LIN {X 0,Y 518.163,Z 728.095,A -85,B 0,C 180,E1 -4999.763,E2 -4999.763} C_VEL
LIN {X 0,Y 517.896,Z 738.556,A -85,B 0,C 180,E1 -5000.474,E2 -5000.474} C_VEL
LIN {X 0,Y 517.639,Z 748.894,A -85,B 0,C 180,E1 -5001.351,E2 -5001.351} C_VEL
LIN {X 0,Y 517.372,Z 758.155,A -85,B 0,C 180,E1 -5002.317,E2 -5002.317} C_VEL
LIN {X 0,Y 517.046,Z 767.447,A -85,B 0,C 180,E1 -5003.531,E2 -5003.531} C_VEL
LIN {X 0,Y 516.894,Z 774.412,A -85,B 0,C 180,E1 -5004.667,E2 -5004.667} C_VEL
LIN {X 0,Y 516.72,Z 779.315,A -85,B 0,C 180,E1 -5005.636,E2 -5005.636} C_VEL
LIN {X 0,Y 516.615,Z 783.22,A -85,B 0,C 180,E1 -5006.567,E2 -5006.567} C_VEL
LIN {X 0,Y 516.59,Z 786.474,A -85,B 0,C 180,E1 -5007.511,E2 -5007.511} C_VEL
LIN {X 0,Y 516.499,Z 789.918,A -85,B 0,C 180,E1 -5008.864,E2 -5008.864} C_VEL
LIN {X 0,Y 516.448,Z 791.553,A -85,B 0,C 180,E1 -5009.767,E2 -5009.767} C_VEL
LIN {X 0,Y 516.407,Z 792.613,A -85,B 0,C 180,E1 -5010.663,E2 -5010.663} C_VEL
LIN {X 0,Y 516.396,Z 793.257,A -85,B 0,C 180,E1 -5012.207,E2 -5012.207} C_VEL
LIN {X 0,Y 516.435,Z 792.788,A -85,B 0,C 180,E1 -5013.315,E2 -5013.315} C_VEL
LIN {X 0,Y 516.442,Z 791.847,A -85,B 0,C 180,E1 -5014.184,E2 -5014.184} C_VEL
LIN {X 0,Y 516.562,Z 789.005,A -85,B 0,C 180,E1 -5015.722,E2 -5015.722} C_VEL
LIN {X 0,Y 516.653,Z 784.693,A -85,B 0,C 180,E1 -5017.189,E2 -5017.189} C_VEL
LIN {X 0,Y 516.772,Z 779.621,A -85,B 0,C 180,E1 -5018.457,E2 -5018.457} C_VEL
LIN {X 0,Y 516.959,Z 774.001,A -85,B 0,C 180,E1 -5019.569,E2 -5019.569} C_VEL
LIN {X 0,Y 517.22,Z 766.534,A -85,B 0,C 180,E1 -5020.761,E2 -5020.761} C_VEL
LIN {X 0,Y 517.462,Z 757.238,A -85,B 0,C 180,E1 -5021.938,E2 -5021.938} C_VEL
LIN {X 0,Y 517.742,Z 747.459,A -85,B 0,C 180,E1 -5022.93,E2 -5022.93} C_VEL
LIN {X 0,Y 518.011,Z 737.439,A -85,B 0,C 180,E1 -5023.75,E2 -5023.75} C_VEL
LIN {X 0,Y 518.228,Z 727.164,A -85,B 0,C 180,E1 -5024.43,E2 -5024.43} C_VEL
LIN {X 0,Y 518.371,Z 718.099,A -85,B 0,C 180,E1 -5024.913,E2 -5024.913} C_VEL
LIN {X 0,Y 516.951,Z 712.094,A -85,B 0,C 180,E1 -5025.232,E2 -5025.232} C_VEL
LIN {X 0,Y 516.971,Z 712.089,A -85,B 0,C 180,E1 -5028.234,E2 -5028.234} C_VEL
LIN {X 0,Y 516.968,Z 712.091,A -85,B 0,C 180,E1 -5031.4,E2 -5031.4} C_VEL
LIN {X 0,Y 517.017,Z 712.078,A -85,B 0,C 180,E1 -5034.54,E2 -5034.54} C_VEL
LIN {X 0,Y 517.085,Z 712.078,A -85,B 0,C 180,E1 -5037.663,E2 -5037.663} C_VEL
LIN {X 0,Y 517.095,Z 712.068,A -85,B 0,C 180,E1 -5040.779,E2 -5040.779} C_VEL
LIN {X 0,Y 516.988,Z 712.08,A -85,B 0,C 180,E1 -5043.117,E2 -5043.117} C_VEL
LIN {X 0,Y 517.013,Z 712.083,A -85,B 0,C 180,E1 -5046.243,E2 -5046.243} C_VEL
LIN {X 0,Y 516.946,Z 712.086,A -85,B 0,C 180,E1 -5049.389,E2 -5049.389} C_VEL
LIN {X 0,Y 516.957,Z 712.091,A -85,B 0,C 180,E1 -5051.807,E2 -5051.807} C_VEL
LIN {X 0,Y 516.949,Z 712.084,A -85,B 0,C 180,E1 -5055.146,E2 -5055.146} C_VEL
LIN {X 0,Y 516.92,Z 712.096,A -85,B 0,C 180,E1 -5058.222,E2 -5058.222} C_VEL
LIN {X 0,Y 516.917,Z 712.091,A -85,B 0,C 180,E1 -5060.701,E2 -5060.701} C_VEL
LIN {X 0,Y 516.895,Z 712.099,A -85,B 0,C 180,E1 -5064.073,E2 -5064.073} C_VEL
LIN {X 0,Y 516.928,Z 712.094,A -85,B 0,C 180,E1 -5066.658,E2 -5066.658} C_VEL
LIN {X 0,Y 516.915,Z 712.091,A -85,B 0,C 180,E1 -5069.524,E2 -5069.524} C_VEL
LIN {X 0,Y 516.902,Z 712.1,A -85,B 0,C 180,E1 -5072.544,E2 -5072.544} C_VEL
LIN {X 0,Y 516.871,Z 712.098,A -85,B 0,C 180,E1 -5075.33,E2 -5075.33} C_VEL
LIN {X 0,Y 516.885,Z 712.099,A -85,B 0,C 180,E1 -5077.943,E2 -5077.943} C_VEL
LIN {X 0,Y 516.888,Z 712.104,A -85,B 0,C 180,E1 -5080.741,E2 -5080.741} C_VEL
LIN {X 0,Y 516.887,Z 712.102,A -85,B 0,C 180,E1 -5082.831,E2 -5082.831} C_VEL
LIN {X 0,Y 516.926,Z 712.095,A -85,B 0,C 180,E1 -5085.01,E2 -5085.01} C_VEL
LIN {X 0,Y 516.92,Z 712.1,A -85,B 0,C 180,E1 -5088.398,E2 -5088.398} C_VEL
LIN {X 0,Y 516.92,Z 712.228,A -85,B 0,C 180,E1 -5091.483,E2 -5091.483} C_VEL
LIN {X 0,Y 518.704,Z 721.914,A -85,B 0,C 180,E1 -5093.886,E2 -5093.886} C_VEL
LIN {X 0,Y 518.509,Z 734.489,A -85,B 0,C 180,E1 -5096.705,E2 -5096.705} C_VEL
LIN {X 0,Y 518.245,Z 748.349,A -85,B 0,C 180,E1 -5099.658,E2 -5099.658} C_VEL
LIN {X 0,Y 518.022,Z 763.378,A -85,B 0,C 180,E1 -5102.749,E2 -5102.749} C_VEL
LIN {X 0,Y 517.836,Z 777.944,A -85,B 0,C 180,E1 -5105.689,E2 -5105.689} C_VEL
LIN {X 0,Y 517.604,Z 794.526,A -85,B 0,C 180,E1 -5108.911,E2 -5108.911} C_VEL
LIN {X 0,Y 517.329,Z 810.368,A -85,B 0,C 180,E1 -5111.983,E2 -5111.983} C_VEL
LIN {X 0,Y 516.966,Z 827.099,A -85,B 0,C 180,E1 -5115.433,E2 -5115.433} C_VEL
LIN {X 0,Y 516.883,Z 830.156,A -85,B 0,C 180,E1 -5116.059,E2 -5116.059} C_VEL
LIN {X 0,Y 518.578,Z 841.514,A -85,B 0,C 180,E1 -5116.33,E2 -5116.33} C_VEL
LIN {X 0,Y 518.347,Z 854.17,A -85,B 0,C 180,E1 -5116.724,E2 -5116.724} C_VEL
LIN {X 0,Y 518.071,Z 866.487,A -85,B 0,C 180,E1 -5117.265,E2 -5117.265} C_VEL
LIN {X 0,Y 517.808,Z 877.914,A -85,B 0,C 180,E1 -5117.928,E2 -5117.928} C_VEL
LIN {X 0,Y 517.521,Z 888.917,A -85,B 0,C 180,E1 -5118.743,E2 -5118.743} C_VEL
LIN {X 0,Y 517.165,Z 898.597,A -85,B 0,C 180,E1 -5119.627,E2 -5119.627} C_VEL
LIN {X 0,Y 516.9,Z 907.411,A -85,B 0,C 180,E1 -5120.61,E2 -5120.61} C_VEL
LIN {X 0,Y 516.683,Z 916.002,A -85,B 0,C 180,E1 -5121.789,E2 -5121.789} C_VEL
LIN {X 0,Y 516.507,Z 922.868,A -85,B 0,C 180,E1 -5122.966,E2 -5122.966} C_VEL
LIN {X 0,Y 516.454,Z 928.365,A -85,B 0,C 180,E1 -5124.142,E2 -5124.142} C_VEL
LIN {X 0,Y 516.271,Z 932.676,A -85,B 0,C 180,E1 -5125.315,E2 -5125.315} C_VEL
LIN {X 0,Y 516.355,Z 934.958,A -85,B 0,C 180,E1 -5126.098,E2 -5126.098} C_VEL
LIN {X 0,Y 516.282,Z 936.807,A -85,B 0,C 180,E1 -5126.879,E2 -5126.879} C_VEL
LIN {X 0,Y 516.26,Z 938.194,A -85,B 0,C 180,E1 -5127.659,E2 -5127.659} C_VEL
LIN {X 0,Y 516.16,Z 939.786,A -85,B 0,C 180,E1 -5129.22,E2 -5129.22} C_VEL
LIN {X 0,Y 516.154,Z 940,A -85,B 0,C 180,E1 -5130,E2 -5130} C_VEL
LIN {X 0,Y 516.191,Z 939.184,A -85,B 0,C 180,E1 -5131.56,E2 -5131.56} C_VEL
LIN {X 0,Y 516.26,Z 938.197,A -85,B 0,C 180,E1 -5132.341,E2 -5132.341} C_VEL
LIN {X 0,Y 516.282,Z 936.81,A -85,B 0,C 180,E1 -5133.121,E2 -5133.121} C_VEL
LIN {X 0,Y 516.343,Z 933.896,A -85,B 0,C 180,E1 -5134.293,E2 -5134.293} C_VEL
LIN {X 0,Y 516.405,Z 929.949,A -85,B 0,C 180,E1 -5135.467,E2 -5135.467} C_VEL
LIN {X 0,Y 516.486,Z 924.033,A -85,B 0,C 180,E1 -5136.807,E2 -5136.807} C_VEL
LIN {X 0,Y 516.641,Z 917.236,A -85,B 0,C 180,E1 -5138.015,E2 -5138.015} C_VEL
LIN {X 0,Y 516.867,Z 908.992,A -85,B 0,C 180,E1 -5139.193,E2 -5139.193} C_VEL
LIN {X 0,Y 517.078,Z 900.54,A -85,B 0,C 180,E1 -5140.177,E2 -5140.177} C_VEL
LIN {X 0,Y 517.484,Z 890.093,A -85,B 0,C 180,E1 -5141.159,E2 -5141.159} C_VEL
LIN {X 0,Y 517.767,Z 879.202,A -85,B 0,C 180,E1 -5141.985,E2 -5141.985} C_VEL
LIN {X 0,Y 517.985,Z 868.405,A -85,B 0,C 180,E1 -5142.638,E2 -5142.638} C_VEL
LIN {X 0,Y 518.298,Z 856.764,A -85,B 0,C 180,E1 -5143.178,E2 -5143.178} C_VEL
LIN {X 0,Y 518.521,Z 844.259,A -85,B 0,C 180,E1 -5143.596,E2 -5143.596} C_VEL
LIN {X 0,Y 518.292,Z 839.065,A -85,B 0,C 180,E1 -5143.734,E2 -5143.734} C_VEL
LIN {X 0,Y 516.879,Z 830.034,A -85,B 0,C 180,E1 -5143.966,E2 -5143.966} C_VEL
LIN {X 0,Y 517.193,Z 815.361,A -85,B 0,C 180,E1 -5146.987,E2 -5146.987} C_VEL
LIN {X 0,Y 517.417,Z 803.193,A -85,B 0,C 180,E1 -5149.438,E2 -5149.438} C_VEL
LIN {X 0,Y 517.661,Z 789.594,A -85,B 0,C 180,E1 -5152.132,E2 -5152.132} C_VEL
LIN {X 0,Y 517.969,Z 776.156,A -85,B 0,C 180,E1 -5154.874,E2 -5154.874} C_VEL
LIN {X 0,Y 518.253,Z 762.094,A -85,B 0,C 180,E1 -5157.821,E2 -5157.821} C_VEL
LIN {X 0,Y 518.621,Z 748.41,A -85,B 0,C 180,E1 -5160.768,E2 -5160.768} C_VEL
LIN {X 0,Y 519.008,Z 735.047,A -85,B 0,C 180,E1 -5163.724,E2 -5163.724} C_VEL
LIN {X 0,Y 519.206,Z 723.868,A -85,B 0,C 180,E1 -5166.313,E2 -5166.313} C_VEL
LIN {X 0,Y 517.688,Z 715.93,A -85,B 0,C 180,E1 -5168.317,E2 -5168.317} C_VEL
LIN {X 0,Y 516.924,Z 712.098,A -85,B 0,C 180,E1 -5169.314,E2 -5169.314} C_VEL
LIN {X 0,Y 516.918,Z 712.096,A -85,B 0,C 180,E1 -5171.775,E2 -5171.775} C_VEL
LIN {X 0,Y 516.925,Z 712.095,A -85,B 0,C 180,E1 -5175.01,E2 -5175.01} C_VEL
LIN {X 0,Y 516.918,Z 712.091,A -85,B 0,C 180,E1 -5178.398,E2 -5178.398} C_VEL
LIN {X 0,Y 516.885,Z 712.102,A -85,B 0,C 180,E1 -5181.284,E2 -5181.284} C_VEL
LIN {X 0,Y 516.874,Z 712.096,A -85,B 0,C 180,E1 -5184.22,E2 -5184.22} C_VEL
LIN {X 0,Y 516.899,Z 712.095,A -85,B 0,C 180,E1 -5187.053,E2 -5187.053} C_VEL
LIN {X 0,Y 516.895,Z 712.1,A -85,B 0,C 180,E1 -5189.796,E2 -5189.796} C_VEL
LIN {X 0,Y 516.929,Z 712.089,A -85,B 0,C 180,E1 -5192.467,E2 -5192.467} C_VEL
LIN {X 0,Y 516.878,Z 712.097,A -85,B 0,C 180,E1 -5195.07,E2 -5195.07} C_VEL
LIN {X 0,Y 516.871,Z 712.103,A -85,B 0,C 180,E1 -5197.622,E2 -5197.622} C_VEL
LIN {X 0,Y 516.934,Z 712.093,A -85,B 0,C 180,E1 -5200.13,E2 -5200.13} C_VEL
LIN {X 0,Y 516.91,Z 712.092,A -85,B 0,C 180,E1 -5202.595,E2 -5202.595} C_VEL
LIN {X 0,Y 516.946,Z 712.088,A -85,B 0,C 180,E1 -5205.03,E2 -5205.03} C_VEL
LIN {X 0,Y 516.969,Z 712.089,A -85,B 0,C 180,E1 -5208.234,E2 -5208.234} C_VEL
LIN {X 0,Y 516.967,Z 712.087,A -85,B 0,C 180,E1 -5211.4,E2 -5211.4} C_VEL
LIN {X 0,Y 517.011,Z 712.085,A -85,B 0,C 180,E1 -5213.757,E2 -5213.757} C_VEL
LIN {X 0,Y 517.084,Z 712.074,A -85,B 0,C 180,E1 -5217.663,E2 -5217.663} C_VEL
LIN {X 0,Y 517.091,Z 712.071,A -85,B 0,C 180,E1 -5220.779,E2 -5220.779} C_VEL
LIN {X 0,Y 516.984,Z 712.083,A -85,B 0,C 180,E1 -5223.117,E2 -5223.117} C_VEL
LIN {X 0,Y 516.989,Z 712.089,A -85,B 0,C 180,E1 -5226.244,E2 -5226.244} C_VEL
LIN {X 0,Y 516.943,Z 712.088,A -85,B 0,C 180,E1 -5229.39,E2 -5229.39} C_VEL
LIN {X 0,Y 516.955,Z 712.089,A -85,B 0,C 180,E1 -5231.807,E2 -5231.807} C_VEL
LIN {X 0,Y 516.942,Z 712.089,A -85,B 0,C 180,E1 -5235.144,E2 -5235.144} C_VEL
LIN {X 0,Y 516.915,Z 712.097,A -85,B 0,C 180,E1 -5238.223,E2 -5238.223} C_VEL
LIN {X 0,Y 516.915,Z 712.098,A -85,B 0,C 180,E1 -5240.702,E2 -5240.702} C_VEL
LIN {X 0,Y 516.887,Z 712.098,A -85,B 0,C 180,E1 -5244.073,E2 -5244.073} C_VEL
LIN {X 0,Y 516.839,Z 712.108,A -85,B 0,C 180,E1 -5246.663,E2 -5246.663} C_VEL
LIN {X 0,Y 516.909,Z 712.093,A -85,B 0,C 180,E1 -5249.523,E2 -5249.523} C_VEL
LIN {X 0,Y 516.897,Z 712.1,A -85,B 0,C 180,E1 -5252.543,E2 -5252.543} C_VEL
LIN {X 0,Y 516.862,Z 712.1,A -85,B 0,C 180,E1 -5255.329,E2 -5255.329} C_VEL
LIN {X 0,Y 516.873,Z 712.103,A -85,B 0,C 180,E1 -5258.717,E2 -5258.717} C_VEL
LIN {X 0,Y 516.847,Z 712.101,A -85,B 0,C 180,E1 -5261.782,E2 -5261.782} C_VEL
LIN {X 0,Y 516.898,Z 712.1,A -85,B 0,C 180,E1 -5265.007,E2 -5265.007} C_VEL
LIN {X 0,Y 516.851,Z 712.102,A -85,B 0,C 180,E1 -5268.407,E2 -5268.407} C_VEL
LIN {X 0,Y 516.859,Z 712.1,A -85,B 0,C 180,E1 -5270.28,E2 -5270.28} C_VEL
LIN {X 0,Y 516.19,Z 712.188,A -85,B 0,C 180,E1 -5270.93,E2 -5270.93} C_VEL
LIN {X 0,Y 513.324,Z 712.547,A -85,B 0,C 180,E1 -5271.986,E2 -5271.986} C_VEL
LIN {X 0,Y 510.899,Z 712.848,A -85,B 0,C 180,E1 -5272.836,E2 -5272.836} C_VEL
LIN {X 0,Y 509.857,Z 712.975,A -85,B 0,C 180,E1 -5273.492,E2 -5273.492} C_VEL
LIN {X 0,Y 509.772,Z 712.983,A -85,B 0,C 180,E1 -5273.715,E2 -5273.715} C_VEL
LIN {X 0,Y 509.827,Z 712.977,A -85,B 0,C 180,E1 -5276.537,E2 -5276.537} C_VEL
LIN {X 0,Y 509.807,Z 712.983,A -85,B 0,C 180,E1 -5279.332,E2 -5279.332} C_VEL
LIN {X 0,Y 509.827,Z 712.975,A -85,B 0,C 180,E1 -5282.05,E2 -5282.05} C_VEL
LIN {X 0,Y 509.783,Z 712.982,A -85,B 0,C 180,E1 -5284.699,E2 -5284.699} C_VEL
LIN {X 0,Y 509.828,Z 712.98,A -85,B 0,C 180,E1 -5287.459,E2 -5287.459} C_VEL
LIN {X 0,Y 509.919,Z 712.966,A -85,B 0,C 180,E1 -5289.845,E2 -5289.845} C_VEL
LIN {X 0,Y 509.849,Z 712.978,A -85,B 0,C 180,E1 -5293.174,E2 -5293.174} C_VEL
LIN {X 0,Y 509.849,Z 712.977,A -85,B 0,C 180,E1 -5295.634,E2 -5295.634} C_VEL
LIN {X 0,Y 509.892,Z 712.968,A -85,B 0,C 180,E1 -5298.131,E2 -5298.131} C_VEL
LIN {X 0,Y 509.874,Z 712.974,A -85,B 0,C 180,E1 -5301.279,E2 -5301.279} C_VEL
LIN {X 0,Y 509.92,Z 712.969,A -85,B 0,C 180,E1 -5303.67,E2 -5303.67} C_VEL
LIN {X 0,Y 509.888,Z 712.968,A -85,B 0,C 180,E1 -5306.84,E2 -5306.84} C_VEL
LIN {X 0,Y 509.924,Z 712.963,A -85,B 0,C 180,E1 -5308.421,E2 -5308.421} C_VEL
LIN {X 0,Y 510.037,Z 712.953,A -85,B 0,C 180,E1 -5310,E2 -5310} C_VEL
LIN {X 0,Y 510.045,Z 712.949,A -85,B 0,C 180,E1 -5312.369,E2 -5312.369} C_VEL
LIN {X 0,Y 509.943,Z 712.966,A -85,B 0,C 180,E1 -5315.536,E2 -5315.536} C_VEL
LIN {X 0,Y 509.889,Z 712.967,A -85,B 0,C 180,E1 -5318.721,E2 -5318.721} C_VEL
LIN {X 0,Y 509.909,Z 712.971,A -85,B 0,C 180,E1 -5321.932,E2 -5321.932} C_VEL
LIN {X 0,Y 509.899,Z 712.966,A -85,B 0,C 180,E1 -5325.242,E2 -5325.242} C_VEL
LIN {X 0,Y 509.861,Z 712.973,A -85,B 0,C 180,E1 -5328.484,E2 -5328.484} C_VEL
LIN {X 0,Y 509.854,Z 712.971,A -85,B 0,C 180,E1 -5331.002,E2 -5331.002} C_VEL
LIN {X 0,Y 509.824,Z 712.977,A -85,B 0,C 180,E1 -5333.564,E2 -5333.564} C_VEL
LIN {X 0,Y 509.841,Z 712.977,A -85,B 0,C 180,E1 -5336.362,E2 -5336.362} C_VEL
LIN {X 0,Y 509.854,Z 712.972,A -85,B 0,C 180,E1 -5338.846,E2 -5338.846} C_VEL
LIN {X 0,Y 509.823,Z 712.975,A -85,B 0,C 180,E1 -5341.59,E2 -5341.59} C_VEL
LIN {X 0,Y 509.842,Z 712.979,A -85,B 0,C 180,E1 -5344.414,E2 -5344.414} C_VEL
LIN {X 0,Y 509.821,Z 712.974,A -85,B 0,C 180,E1 -5347.341,E2 -5347.341} C_VEL
LIN {X 0,Y 509.842,Z 712.981,A -85,B 0,C 180,E1 -5350.382,E2 -5350.382} C_VEL
LIN {X 0,Y 509.826,Z 712.975,A -85,B 0,C 180,E1 -5353.062,E2 -5353.062} C_VEL
LIN {X 0,Y 509.826,Z 712.975,A -85,B 0,C 180,E1 -5355.793,E2 -5355.793} C_VEL
LIN {X 0,Y 509.881,Z 712.975,A -85,B 0,C 180,E1 -5358.706,E2 -5358.706} C_VEL
LIN {X 0,Y 511.488,Z 719.855,A -85,B 0,C 180,E1 -5359.089,E2 -5359.089} C_VEL
LIN {X 0,Y 511.22,Z 731.401,A -85,B 0,C 180,E1 -5359.749,E2 -5359.749} C_VEL
LIN {X 0,Y 510.913,Z 742.512,A -85,B 0,C 180,E1 -5360.557,E2 -5360.557} C_VEL
LIN {X 0,Y 510.598,Z 753.016,A -85,B 0,C 180,E1 -5361.524,E2 -5361.524} C_VEL
LIN {X 0,Y 510.361,Z 761.296,A -85,B 0,C 180,E1 -5362.457,E2 -5362.457} C_VEL
LIN {X 0,Y 510.091,Z 768.654,A -85,B 0,C 180,E1 -5363.454,E2 -5363.454} C_VEL
LIN {X 0,Y 509.907,Z 775.719,A -85,B 0,C 180,E1 -5364.628,E2 -5364.628} C_VEL
LIN {X 0,Y 509.713,Z 781.508,A -85,B 0,C 180,E1 -5365.822,E2 -5365.822} C_VEL
LIN {X 0,Y 509.585,Z 786.929,A -85,B 0,C 180,E1 -5367.277,E2 -5367.277} C_VEL
LIN {X 0,Y 509.489,Z 790.877,A -85,B 0,C 180,E1 -5368.787,E2 -5368.787} C_VEL
LIN {X 0,Y 509.405,Z 793.344,A -85,B 0,C 180,E1 -5370.364,E2 -5370.364} C_VEL
LIN {X 0,Y 509.381,Z 794.008,A -85,B 0,C 180,E1 -5371.125,E2 -5371.125} C_VEL
LIN {X 0,Y 509.371,Z 794.314,A -85,B 0,C 180,E1 -5372.023,E2 -5372.023} C_VEL
LIN {X 0,Y 509.397,Z 794.077,A -85,B 0,C 180,E1 -5372.916,E2 -5372.916} C_VEL
LIN {X 0,Y 509.412,Z 793.381,A -85,B 0,C 180,E1 -5373.801,E2 -5373.801} C_VEL
LIN {X 0,Y 509.451,Z 792.213,A -85,B 0,C 180,E1 -5374.681,E2 -5374.681} C_VEL
LIN {X 0,Y 509.587,Z 789.5,A -85,B 0,C 180,E1 -5375.993,E2 -5375.993} C_VEL
LIN {X 0,Y 509.682,Z 785.658,A -85,B 0,C 180,E1 -5377.288,E2 -5377.288} C_VEL
LIN {X 0,Y 509.819,Z 780.566,A -85,B 0,C 180,E1 -5378.573,E2 -5378.573} C_VEL
LIN {X 0,Y 510.037,Z 774.104,A -85,B 0,C 180,E1 -5379.849,E2 -5379.849} C_VEL
LIN {X 0,Y 510.309,Z 765.899,A -85,B 0,C 180,E1 -5381.116,E2 -5381.116} C_VEL
LIN {X 0,Y 510.609,Z 756.887,A -85,B 0,C 180,E1 -5382.231,E2 -5382.231} C_VEL
LIN {X 0,Y 510.882,Z 747.068,A -85,B 0,C 180,E1 -5383.208,E2 -5383.208} C_VEL
LIN {X 0,Y 511.223,Z 735.481,A -85,B 0,C 180,E1 -5384.125,E2 -5384.125} C_VEL
LIN {X 0,Y 511.431,Z 724.883,A -85,B 0,C 180,E1 -5384.789,E2 -5384.789} C_VEL
LIN {X 0,Y 511.534,Z 719.426,A -85,B 0,C 180,E1 -5385.072,E2 -5385.072} C_VEL
LIN {X 0,Y 509.894,Z 712.974,A -85,B 0,C 180,E1 -5385.431,E2 -5385.431} C_VEL
LIN {X 0,Y 509.924,Z 712.968,A -85,B 0,C 180,E1 -5388.114,E2 -5388.114} C_VEL
LIN {X 0,Y 509.914,Z 712.968,A -85,B 0,C 180,E1 -5391.28,E2 -5391.28} C_VEL
LIN {X 0,Y 509.968,Z 712.957,A -85,B 0,C 180,E1 -5394.464,E2 -5394.464} C_VEL
LIN {X 0,Y 510.054,Z 712.954,A -85,B 0,C 180,E1 -5397.631,E2 -5397.631} C_VEL
LIN {X 0,Y 510.066,Z 712.944,A -85,B 0,C 180,E1 -5400.789,E2 -5400.789} C_VEL
LIN {X 0,Y 509.932,Z 712.959,A -85,B 0,C 180,E1 -5403.16,E2 -5403.16} C_VEL
LIN {X 0,Y 509.963,Z 712.96,A -85,B 0,C 180,E1 -5406.33,E2 -5406.33} C_VEL
LIN {X 0,Y 509.887,Z 712.966,A -85,B 0,C 180,E1 -5409.521,E2 -5409.521} C_VEL
LIN {X 0,Y 509.909,Z 712.969,A -85,B 0,C 180,E1 -5411.932,E2 -5411.932} C_VEL
LIN {X 0,Y 509.899,Z 712.962,A -85,B 0,C 180,E1 -5415.242,E2 -5415.242} C_VEL
LIN {X 0,Y 509.871,Z 712.975,A -85,B 0,C 180,E1 -5417.993,E2 -5417.993} C_VEL
LIN {X 0,Y 509.891,Z 712.97,A -85,B 0,C 180,E1 -5420.401,E2 -5420.401} C_VEL
LIN {X 0,Y 509.826,Z 712.974,A -85,B 0,C 180,E1 -5423.564,E2 -5423.564} C_VEL
LIN {X 0,Y 509.915,Z 712.969,A -85,B 0,C 180,E1 -5426.378,E2 -5426.378} C_VEL
LIN {X 0,Y 509.88,Z 712.97,A -85,B 0,C 180,E1 -5428.844,E2 -5428.844} C_VEL
LIN {X 0,Y 509.825,Z 712.974,A -85,B 0,C 180,E1 -5431.59,E2 -5431.59} C_VEL
LIN {X 0,Y 509.852,Z 712.98,A -85,B 0,C 180,E1 -5434.414,E2 -5434.414} C_VEL
LIN {X 0,Y 509.82,Z 712.978,A -85,B 0,C 180,E1 -5437.341,E2 -5437.341} C_VEL
LIN {X 0,Y 509.842,Z 712.981,A -85,B 0,C 180,E1 -5440.382,E2 -5440.382} C_VEL
LIN {X 0,Y 509.827,Z 712.979,A -85,B 0,C 180,E1 -5443.062,E2 -5443.062} C_VEL
LIN {X 0,Y 509.834,Z 712.975,A -85,B 0,C 180,E1 -5445.792,E2 -5445.792} C_VEL
LIN {X 0,Y 509.862,Z 712.979,A -85,B 0,C 180,E1 -5448.575,E2 -5448.575} C_VEL
LIN {X 0,Y 509.872,Z 713.052,A -85,B 0,C 180,E1 -5451.222,E2 -5451.222} C_VEL
LIN {X 0,Y 511.515,Z 721.365,A -85,B 0,C 180,E1 -5453.354,E2 -5453.354} C_VEL
LIN {X 0,Y 511.723,Z 725.952,A -85,B 0,C 180,E1 -5454.445,E2 -5454.445} C_VEL
LIN {X 0,Y 511.472,Z 738.499,A -85,B 0,C 180,E1 -5457.269,E2 -5457.269} C_VEL
LIN {X 0,Y 511.187,Z 751.219,A -85,B 0,C 180,E1 -5460.014,E2 -5460.014} C_VEL
LIN {X 0,Y 510.992,Z 765.578,A -85,B 0,C 180,E1 -5463.007,E2 -5463.007} C_VEL
LIN {X 0,Y 510.72,Z 780.468,A -85,B 0,C 180,E1 -5466.049,E2 -5466.049} C_VEL
LIN {X 0,Y 510.507,Z 795.562,A -85,B 0,C 180,E1 -5469.026,E2 -5469.026} C_VEL
LIN {X 0,Y 510.195,Z 812.615,A -85,B 0,C 180,E1 -5472.359,E2 -5472.359} C_VEL
LIN {X 0,Y 509.925,Z 827.099,A -85,B 0,C 180,E1 -5475.228,E2 -5475.228} C_VEL
LIN {X 0,Y 509.852,Z 830.155,A -85,B 0,C 180,E1 -5475.863,E2 -5475.863} C_VEL
LIN {X 0,Y 511.659,Z 842.429,A -85,B 0,C 180,E1 -5476.167,E2 -5476.167} C_VEL
LIN {X 0,Y 511.419,Z 855.47,A -85,B 0,C 180,E1 -5476.591,E2 -5476.591} C_VEL
LIN {X 0,Y 511.143,Z 866.486,A -85,B 0,C 180,E1 -5477.089,E2 -5477.089} C_VEL
LIN {X 0,Y 510.827,Z 877.914,A -85,B 0,C 180,E1 -5477.76,E2 -5477.76} C_VEL
LIN {X 0,Y 510.551,Z 888.916,A -85,B 0,C 180,E1 -5478.587,E2 -5478.587} C_VEL
LIN {X 0,Y 510.173,Z 898.596,A -85,B 0,C 180,E1 -5479.483,E2 -5479.483} C_VEL
LIN {X 0,Y 509.887,Z 907.411,A -85,B 0,C 180,E1 -5480.479,E2 -5480.479} C_VEL
LIN {X 0,Y 509.624,Z 916.003,A -85,B 0,C 180,E1 -5481.674,E2 -5481.674} C_VEL
LIN {X 0,Y 509.422,Z 922.867,A -85,B 0,C 180,E1 -5482.867,E2 -5482.867} C_VEL
LIN {X 0,Y 509.368,Z 928.365,A -85,B 0,C 180,E1 -5484.06,E2 -5484.06} C_VEL
LIN {X 0,Y 509.188,Z 932.676,A -85,B 0,C 180,E1 -5485.25,E2 -5485.25} C_VEL
LIN {X 0,Y 509.253,Z 934.958,A -85,B 0,C 180,E1 -5486.043,E2 -5486.043} C_VEL
LIN {X 0,Y 509.201,Z 936.807,A -85,B 0,C 180,E1 -5486.835,E2 -5486.835} C_VEL
LIN {X 0,Y 509.16,Z 938.194,A -85,B 0,C 180,E1 -5487.627,E2 -5487.627} C_VEL
LIN {X 0,Y 509.073,Z 939.786,A -85,B 0,C 180,E1 -5489.209,E2 -5489.209} C_VEL
LIN {X 0,Y 509.065,Z 940,A -85,B 0,C 180,E1 -5490,E2 -5490} C_VEL
LIN {X 0,Y 509.112,Z 939.184,A -85,B 0,C 180,E1 -5491.582,E2 -5491.582} C_VEL
LIN {X 0,Y 509.16,Z 938.196,A -85,B 0,C 180,E1 -5492.373,E2 -5492.373} C_VEL
LIN {X 0,Y 509.201,Z 936.81,A -85,B 0,C 180,E1 -5493.165,E2 -5493.165} C_VEL
LIN {X 0,Y 509.234,Z 933.896,A -85,B 0,C 180,E1 -5494.353,E2 -5494.353} C_VEL
LIN {X 0,Y 509.344,Z 929.948,A -85,B 0,C 180,E1 -5495.543,E2 -5495.543} C_VEL
LIN {X 0,Y 509.41,Z 924.281,A -85,B 0,C 180,E1 -5496.853,E2 -5496.853} C_VEL
LIN {X 0,Y 509.585,Z 917.236,A -85,B 0,C 180,E1 -5498.127,E2 -5498.127} C_VEL
LIN {X 0,Y 509.846,Z 908.992,A -85,B 0,C 180,E1 -5499.321,E2 -5499.321} C_VEL
LIN {X 0,Y 510.067,Z 900.54,A -85,B 0,C 180,E1 -5500.319,E2 -5500.319} C_VEL
LIN {X 0,Y 510.508,Z 890.091,A -85,B 0,C 180,E1 -5501.313,E2 -5501.313} C_VEL
LIN {X 0,Y 510.853,Z 878.916,A -85,B 0,C 180,E1 -5502.17,E2 -5502.17} C_VEL
LIN {X 0,Y 511.053,Z 868.404,A -85,B 0,C 180,E1 -5502.812,E2 -5502.812} C_VEL
LIN {X 0,Y 511.385,Z 856.764,A -85,B 0,C 180,E1 -5503.359,E2 -5503.359} C_VEL
LIN {X 0,Y 511.65,Z 843.344,A -85,B 0,C 180,E1 -5503.808,E2 -5503.808} C_VEL
LIN {X 0,Y 510.799,Z 836.076,A -85,B 0,C 180,E1 -5504.006,E2 -5504.006} C_VEL
LIN {X 0,Y 509.865,Z 830.034,A -85,B 0,C 180,E1 -5504.162,E2 -5504.162} C_VEL
LIN {X 0,Y 510.138,Z 815.895,A -85,B 0,C 180,E1 -5507.023,E2 -5507.023} C_VEL
LIN {X 0,Y 510.4,Z 801.367,A -85,B 0,C 180,E1 -5509.925,E2 -5509.925} C_VEL
LIN {X 0,Y 510.703,Z 787.25,A -85,B 0,C 180,E1 -5512.777,E2 -5512.777} C_VEL
LIN {X 0,Y 511.049,Z 772.439,A -85,B 0,C 180,E1 -5515.889,E2 -5515.889} C_VEL
LIN {X 0,Y 511.326,Z 759.053,A -85,B 0,C 180,E1 -5518.755,E2 -5518.755} C_VEL
LIN {X 0,Y 511.746,Z 746.052,A -85,B 0,C 180,E1 -5521.628,E2 -5521.628} C_VEL
LIN {X 0,Y 512.108,Z 734.534,A -85,B 0,C 180,E1 -5524.241,E2 -5524.241} C_VEL
LIN {X 0,Y 512.309,Z 725.361,A -85,B 0,C 180,E1 -5526.393,E2 -5526.393} C_VEL
LIN {X 0,Y 510.472,Z 716.087,A -85,B 0,C 180,E1 -5528.787,E2 -5528.787} C_VEL
LIN {X 0,Y 509.863,Z 712.977,A -85,B 0,C 180,E1 -5529.649,E2 -5529.649} C_VEL
LIN {X 0,Y 509.837,Z 712.976,A -85,B 0,C 180,E1 -5532.49,E2 -5532.49} C_VEL
LIN {X 0,Y 509.859,Z 712.977,A -85,B 0,C 180,E1 -5535.332,E2 -5535.332} C_VEL
LIN {X 0,Y 509.86,Z 712.971,A -85,B 0,C 180,E1 -5538.575,E2 -5538.575} C_VEL
LIN {X 0,Y 509.854,Z 712.975,A -85,B 0,C 180,E1 -5541.786,E2 -5541.786} C_VEL
LIN {X 0,Y 509.833,Z 712.973,A -85,B 0,C 180,E1 -5544.622,E2 -5544.622} C_VEL
LIN {X 0,Y 509.866,Z 712.976,A -85,B 0,C 180,E1 -5547.481,E2 -5547.481} C_VEL
LIN {X 0,Y 509.861,Z 712.971,A -85,B 0,C 180,E1 -5550.274,E2 -5550.274} C_VEL
LIN {X 0,Y 509.886,Z 712.967,A -85,B 0,C 180,E1 -5552.944,E2 -5552.944} C_VEL
LIN {X 0,Y 509.854,Z 712.977,A -85,B 0,C 180,E1 -5555.573,E2 -5555.573} C_VEL
LIN {X 0,Y 509.824,Z 712.978,A -85,B 0,C 180,E1 -5558.149,E2 -5558.149} C_VEL
LIN {X 0,Y 509.865,Z 712.97,A -85,B 0,C 180,E1 -5560.682,E2 -5560.682} C_VEL
LIN {X 0,Y 509.878,Z 712.969,A -85,B 0,C 180,E1 -5563.175,E2 -5563.175} C_VEL
LIN {X 0,Y 509.866,Z 712.974,A -85,B 0,C 180,E1 -5565.634,E2 -5565.634} C_VEL
LIN {X 0,Y 509.916,Z 712.963,A -85,B 0,C 180,E1 -5568.875,E2 -5568.875} C_VEL
LIN {X 0,Y 509.954,Z 712.967,A -85,B 0,C 180,E1 -5572.079,E2 -5572.079} C_VEL
LIN {X 0,Y 509.982,Z 712.958,A -85,B 0,C 180,E1 -5574.464,E2 -5574.464} C_VEL
LIN {X 0,Y 510.053,Z 712.95,A -85,B 0,C 180,E1 -5577.631,E2 -5577.631} C_VEL
LIN {X 0,Y 510.06,Z 712.951,A -85,B 0,C 180,E1 -5580,E2 -5580} C_VEL
LIN {X 0,Y 510.053,Z 712.953,A -85,B 0,C 180,E1 -5582.369,E2 -5582.369} C_VEL
LIN {X 0,Y 509.971,Z 712.958,A -85,B 0,C 180,E1 -5585.536,E2 -5585.536} C_VEL
LIN {X 0,Y 509.912,Z 712.967,A -85,B 0,C 180,E1 -5588.72,E2 -5588.72} C_VEL
LIN {X 0,Y 509.907,Z 712.969,A -85,B 0,C 180,E1 -5591.932,E2 -5591.932} C_VEL
LIN {X 0,Y 509.897,Z 712.966,A -85,B 0,C 180,E1 -5595.242,E2 -5595.242} C_VEL
LIN {X 0,Y 509.859,Z 712.977,A -85,B 0,C 180,E1 -5598.484,E2 -5598.484} C_VEL
LIN {X 0,Y 509.853,Z 712.974,A -85,B 0,C 180,E1 -5601.002,E2 -5601.002} C_VEL
LIN {X 0,Y 509.821,Z 712.976,A -85,B 0,C 180,E1 -5603.564,E2 -5603.564} C_VEL
LIN {X 0,Y 509.81,Z 712.982,A -85,B 0,C 180,E1 -5606.355,E2 -5606.355} C_VEL
LIN {X 0,Y 509.851,Z 712.978,A -85,B 0,C 180,E1 -5608.846,E2 -5608.846} C_VEL
LIN {X 0,Y 509.82,Z 712.976,A -85,B 0,C 180,E1 -5611.59,E2 -5611.59} C_VEL
LIN {X 0,Y 509.837,Z 712.979,A -85,B 0,C 180,E1 -5614.415,E2 -5614.415} C_VEL
LIN {X 0,Y 509.795,Z 712.981,A -85,B 0,C 180,E1 -5617.343,E2 -5617.343} C_VEL
LIN {X 0,Y 509.815,Z 712.98,A -85,B 0,C 180,E1 -5620.385,E2 -5620.385} C_VEL
LIN {X 0,Y 509.807,Z 712.979,A -85,B 0,C 180,E1 -5623.574,E2 -5623.574} C_VEL
LIN {X 0,Y 509.807,Z 712.98,A -85,B 0,C 180,E1 -5626.427,E2 -5626.427} C_VEL
LIN {X 0,Y 509.814,Z 712.978,A -85,B 0,C 180,E1 -5629.615,E2 -5629.615} C_VEL
LIN {X 0,Y 509.784,Z 712.984,A -85,B 0,C 180,E1 -5632.656,E2 -5632.656} C_VEL
LIN {X 0,Y 509.772,Z 712.983,A -85,B 0,C 180,E1 -5633.715,E2 -5633.715} C_VEL
LIN {X 0,Y 509.112,Z 713.066,A -85,B 0,C 180,E1 -5634.375,E2 -5634.375} C_VEL
LIN {X 0,Y 506.287,Z 713.421,A -85,B 0,C 180,E1 -5635.447,E2 -5635.447} C_VEL
LIN {X 0,Y 503.891,Z 713.722,A -85,B 0,C 180,E1 -5636.311,E2 -5636.311} C_VEL
LIN {X 0,Y 502.849,Z 713.85,A -85,B 0,C 180,E1 -5636.977,E2 -5636.977} C_VEL
LIN {X 0,Y 502.758,Z 713.859,A -85,B 0,C 180,E1 -5637.203,E2 -5637.203} C_VEL
LIN {X 0,Y 502.792,Z 713.852,A -85,B 0,C 180,E1 -5640.07,E2 -5640.07} C_VEL
LIN {X 0,Y 502.771,Z 713.855,A -85,B 0,C 180,E1 -5642.529,E2 -5642.529} C_VEL
LIN {X 0,Y 502.764,Z 713.86,A -85,B 0,C 180,E1 -5645.316,E2 -5645.316} C_VEL
LIN {X 0,Y 502.782,Z 713.855,A -85,B 0,C 180,E1 -5647.826,E2 -5647.826} C_VEL
LIN {X 0,Y 502.821,Z 713.848,A -85,B 0,C 180,E1 -5650.4,E2 -5650.4} C_VEL
LIN {X 0,Y 502.796,Z 713.854,A -85,B 0,C 180,E1 -5652.93,E2 -5652.93} C_VEL
LIN {X 0,Y 502.829,Z 713.852,A -85,B 0,C 180,E1 -5655.429,E2 -5655.429} C_VEL
LIN {X 0,Y 502.838,Z 713.846,A -85,B 0,C 180,E1 -5658.716,E2 -5658.716} C_VEL
LIN {X 0,Y 502.849,Z 713.848,A -85,B 0,C 180,E1 -5661.966,E2 -5661.966} C_VEL
LIN {X 0,Y 502.895,Z 713.839,A -85,B 0,C 180,E1 -5664.386,E2 -5664.386} C_VEL
LIN {X 0,Y 503.011,Z 713.83,A -85,B 0,C 180,E1 -5667.598,E2 -5667.598} C_VEL
LIN {X 0,Y 503.006,Z 713.829,A -85,B 0,C 180,E1 -5670,E2 -5670} C_VEL
LIN {X 0,Y 503.012,Z 713.825,A -85,B 0,C 180,E1 -5672.402,E2 -5672.402} C_VEL
LIN {X 0,Y 502.9,Z 713.844,A -85,B 0,C 180,E1 -5675.614,E2 -5675.614} C_VEL
LIN {X 0,Y 502.853,Z 713.848,A -85,B 0,C 180,E1 -5678.034,E2 -5678.034} C_VEL
LIN {X 0,Y 502.88,Z 713.841,A -85,B 0,C 180,E1 -5681.283,E2 -5681.283} C_VEL
LIN {X 0,Y 502.847,Z 713.845,A -85,B 0,C 180,E1 -5684.571,E2 -5684.571} C_VEL
LIN {X 0,Y 502.821,Z 713.855,A -85,B 0,C 180,E1 -5687.909,E2 -5687.909} C_VEL
LIN {X 0,Y 502.833,Z 713.848,A -85,B 0,C 180,E1 -5690.536,E2 -5690.536} C_VEL
LIN {X 0,Y 502.791,Z 713.851,A -85,B 0,C 180,E1 -5693.041,E2 -5693.041} C_VEL
LIN {X 0,Y 502.785,Z 713.854,A -85,B 0,C 180,E1 -5695.679,E2 -5695.679} C_VEL
LIN {X 0,Y 502.799,Z 713.855,A -85,B 0,C 180,E1 -5698.375,E2 -5698.375} C_VEL
LIN {X 0,Y 502.798,Z 713.849,A -85,B 0,C 180,E1 -5701.143,E2 -5701.143} C_VEL
LIN {X 0,Y 502.793,Z 713.855,A -85,B 0,C 180,E1 -5703.995,E2 -5703.995} C_VEL
LIN {X 0,Y 502.782,Z 713.852,A -85,B 0,C 180,E1 -5707.178,E2 -5707.178} C_VEL
LIN {X 0,Y 502.792,Z 713.854,A -85,B 0,C 180,E1 -5710.015,E2 -5710.015} C_VEL
LIN {X 0,Y 502.807,Z 713.854,A -85,B 0,C 180,E1 -5712.199,E2 -5712.199} C_VEL
LIN {X 0,Y 502.789,Z 713.851,A -85,B 0,C 180,E1 -5715.47,E2 -5715.47} C_VEL
LIN {X 0,Y 502.829,Z 713.862,A -85,B 0,C 180,E1 -5718.527,E2 -5718.527} C_VEL
LIN {X 0,Y 504.598,Z 721.14,A -85,B 0,C 180,E1 -5718.933,E2 -5718.933} C_VEL
LIN {X 0,Y 504.316,Z 733.501,A -85,B 0,C 180,E1 -5719.66,E2 -5719.66} C_VEL
LIN {X 0,Y 503.953,Z 744.406,A -85,B 0,C 180,E1 -5720.485,E2 -5720.485} C_VEL
LIN {X 0,Y 503.679,Z 754.838,A -85,B 0,C 180,E1 -5721.476,E2 -5721.476} C_VEL
LIN {X 0,Y 503.392,Z 763.654,A -85,B 0,C 180,E1 -5722.507,E2 -5722.507} C_VEL
LIN {X 0,Y 503.106,Z 771.191,A -85,B 0,C 180,E1 -5723.58,E2 -5723.58} C_VEL
LIN {X 0,Y 502.906,Z 778.195,A -85,B 0,C 180,E1 -5724.813,E2 -5724.813} C_VEL
LIN {X 0,Y 502.704,Z 783.584,A -85,B 0,C 180,E1 -5725.998,E2 -5725.998} C_VEL
LIN {X 0,Y 502.567,Z 788.711,A -85,B 0,C 180,E1 -5727.468,E2 -5727.468} C_VEL
LIN {X 0,Y 502.466,Z 792.072,A -85,B 0,C 180,E1 -5728.834,E2 -5728.834} C_VEL
LIN {X 0,Y 502.403,Z 794.164,A -85,B 0,C 180,E1 -5730.147,E2 -5730.147} C_VEL
LIN {X 0,Y 502.371,Z 795.244,A -85,B 0,C 180,E1 -5731.598,E2 -5731.598} C_VEL
LIN {X 0,Y 502.37,Z 795.29,A -85,B 0,C 180,E1 -5732.505,E2 -5732.505} C_VEL
LIN {X 0,Y 502.389,Z 794.701,A -85,B 0,C 180,E1 -5733.549,E2 -5733.549} C_VEL
LIN {X 0,Y 502.42,Z 793.87,A -85,B 0,C 180,E1 -5734.301,E2 -5734.301} C_VEL
LIN {X 0,Y 502.516,Z 792.073,A -85,B 0,C 180,E1 -5735.377,E2 -5735.377} C_VEL
LIN {X 0,Y 502.659,Z 788.07,A -85,B 0,C 180,E1 -5736.953,E2 -5736.953} C_VEL
LIN {X 0,Y 502.813,Z 783.389,A -85,B 0,C 180,E1 -5738.259,E2 -5738.259} C_VEL
LIN {X 0,Y 503.014,Z 777.325,A -85,B 0,C 180,E1 -5739.556,E2 -5739.556} C_VEL
LIN {X 0,Y 503.313,Z 769.688,A -85,B 0,C 180,E1 -5740.844,E2 -5740.844} C_VEL
LIN {X 0,Y 503.585,Z 761.497,A -85,B 0,C 180,E1 -5741.956,E2 -5741.956} C_VEL
LIN {X 0,Y 503.935,Z 752.221,A -85,B 0,C 180,E1 -5742.97,E2 -5742.97} C_VEL
LIN {X 0,Y 504.222,Z 741.15,A -85,B 0,C 180,E1 -5743.946,E2 -5743.946} C_VEL
LIN {X 0,Y 504.508,Z 729.446,A -85,B 0,C 180,E1 -5744.755,E2 -5744.755} C_VEL
LIN {X 0,Y 504.553,Z 720.095,A -85,B 0,C 180,E1 -5745.273,E2 -5745.273} C_VEL
LIN {X 0,Y 502.822,Z 713.855,A -85,B 0,C 180,E1 -5745.635,E2 -5745.635} C_VEL
LIN {X 0,Y 502.884,Z 713.843,A -85,B 0,C 180,E1 -5748.717,E2 -5748.717} C_VEL
LIN {X 0,Y 502.884,Z 713.844,A -85,B 0,C 180,E1 -5751.966,E2 -5751.966} C_VEL
LIN {X 0,Y 502.869,Z 713.843,A -85,B 0,C 180,E1 -5755.19,E2 -5755.19} C_VEL
LIN {X 0,Y 503.023,Z 713.83,A -85,B 0,C 180,E1 -5757.598,E2 -5757.598} C_VEL
LIN {X 0,Y 503.015,Z 713.822,A -85,B 0,C 180,E1 -5760.8,E2 -5760.8} C_VEL
LIN {X 0,Y 503.025,Z 713.821,A -85,B 0,C 180,E1 -5762.402,E2 -5762.402} C_VEL
LIN {X 0,Y 502.938,Z 713.837,A -85,B 0,C 180,E1 -5765.613,E2 -5765.613} C_VEL
LIN {X 0,Y 502.884,Z 713.844,A -85,B 0,C 180,E1 -5768.034,E2 -5768.034} C_VEL
LIN {X 0,Y 502.881,Z 713.84,A -85,B 0,C 180,E1 -5771.283,E2 -5771.283} C_VEL
LIN {X 0,Y 502.849,Z 713.843,A -85,B 0,C 180,E1 -5774.571,E2 -5774.571} C_VEL
LIN {X 0,Y 502.845,Z 713.849,A -85,B 0,C 180,E1 -5777.908,E2 -5777.908} C_VEL
LIN {X 0,Y 502.833,Z 713.847,A -85,B 0,C 180,E1 -5780.536,E2 -5780.536} C_VEL
LIN {X 0,Y 502.792,Z 713.85,A -85,B 0,C 180,E1 -5783.041,E2 -5783.041} C_VEL
LIN {X 0,Y 502.825,Z 713.848,A -85,B 0,C 180,E1 -5785.676,E2 -5785.676} C_VEL
LIN {X 0,Y 502.844,Z 713.851,A -85,B 0,C 180,E1 -5788.372,E2 -5788.372} C_VEL
LIN {X 0,Y 502.797,Z 713.85,A -85,B 0,C 180,E1 -5791.499,E2 -5791.499} C_VEL
LIN {X 0,Y 502.808,Z 713.852,A -85,B 0,C 180,E1 -5793.994,E2 -5793.994} C_VEL
LIN {X 0,Y 502.781,Z 713.855,A -85,B 0,C 180,E1 -5797.178,E2 -5797.178} C_VEL
LIN {X 0,Y 502.792,Z 713.856,A -85,B 0,C 180,E1 -5800.015,E2 -5800.015} C_VEL
LIN {X 0,Y 502.806,Z 713.855,A -85,B 0,C 180,E1 -5802.199,E2 -5802.199} C_VEL
LIN {X 0,Y 502.804,Z 713.852,A -85,B 0,C 180,E1 -5805.468,E2 -5805.468} C_VEL
LIN {X 0,Y 502.824,Z 713.855,A -85,B 0,C 180,E1 -5808.934,E2 -5808.934} C_VEL
LIN {X 0,Y 502.807,Z 713.919,A -85,B 0,C 180,E1 -5810.96,E2 -5810.96} C_VEL
LIN {X 0,Y 504.729,Z 723.956,A -85,B 0,C 180,E1 -5813.579,E2 -5813.579} C_VEL
LIN {X 0,Y 504.635,Z 732.949,A -85,B 0,C 180,E1 -5815.697,E2 -5815.697} C_VEL
LIN {X 0,Y 504.363,Z 745.838,A -85,B 0,C 180,E1 -5818.59,E2 -5818.59} C_VEL
LIN {X 0,Y 504.008,Z 761.354,A -85,B 0,C 180,E1 -5821.925,E2 -5821.925} C_VEL
LIN {X 0,Y 503.761,Z 776.448,A -85,B 0,C 180,E1 -5825.07,E2 -5825.07} C_VEL
LIN {X 0,Y 503.488,Z 790.129,A -85,B 0,C 180,E1 -5827.859,E2 -5827.859} C_VEL
LIN {X 0,Y 503.212,Z 805.146,A -85,B 0,C 180,E1 -5830.84,E2 -5830.84} C_VEL
LIN {X 0,Y 502.989,Z 817.853,A -85,B 0,C 180,E1 -5833.355,E2 -5833.355} C_VEL
LIN {X 0,Y 502.825,Z 829.508,A -85,B 0,C 180,E1 -5835.661,E2 -5835.661} C_VEL
LIN {X 0,Y 504.721,Z 842.835,A -85,B 0,C 180,E1 -5835.999,E2 -5835.999} C_VEL
LIN {X 0,Y 504.478,Z 856.419,A -85,B 0,C 180,E1 -5836.454,E2 -5836.454} C_VEL
LIN {X 0,Y 504.123,Z 868.233,A -85,B 0,C 180,E1 -5837.009,E2 -5837.009} C_VEL
LIN {X 0,Y 503.853,Z 879.553,A -85,B 0,C 180,E1 -5837.707,E2 -5837.707} C_VEL
LIN {X 0,Y 503.513,Z 890.089,A -85,B 0,C 180,E1 -5838.527,E2 -5838.527} C_VEL
LIN {X 0,Y 503.063,Z 900.538,A -85,B 0,C 180,E1 -5839.536,E2 -5839.536} C_VEL
LIN {X 0,Y 502.814,Z 908.991,A -85,B 0,C 180,E1 -5840.547,E2 -5840.547} C_VEL
LIN {X 0,Y 502.542,Z 917.234,A -85,B 0,C 180,E1 -5841.758,E2 -5841.758} C_VEL
LIN {X 0,Y 502.346,Z 923.876,A -85,B 0,C 180,E1 -5842.969,E2 -5842.969} C_VEL
LIN {X 0,Y 502.26,Z 929.949,A -85,B 0,C 180,E1 -5844.379,E2 -5844.379} C_VEL
LIN {X 0,Y 502.128,Z 933.894,A -85,B 0,C 180,E1 -5845.585,E2 -5845.585} C_VEL
LIN {X 0,Y 502.121,Z 936.806,A -85,B 0,C 180,E1 -5846.79,E2 -5846.79} C_VEL
LIN {X 0,Y 502.035,Z 939.182,A -85,B 0,C 180,E1 -5848.396,E2 -5848.396} C_VEL
LIN {X 0,Y 501.98,Z 940,A -85,B 0,C 180,E1 -5850,E2 -5850} C_VEL
LIN {X 0,Y 502.035,Z 939.183,A -85,B 0,C 180,E1 -5851.604,E2 -5851.604} C_VEL
LIN {X 0,Y 502.121,Z 936.81,A -85,B 0,C 180,E1 -5853.209,E2 -5853.209} C_VEL
LIN {X 0,Y 502.128,Z 933.895,A -85,B 0,C 180,E1 -5854.415,E2 -5854.415} C_VEL
LIN {X 0,Y 502.259,Z 929.948,A -85,B 0,C 180,E1 -5855.621,E2 -5855.621} C_VEL
LIN {X 0,Y 502.335,Z 923.976,A -85,B 0,C 180,E1 -5857.011,E2 -5857.011} C_VEL
LIN {X 0,Y 502.542,Z 917.235,A -85,B 0,C 180,E1 -5858.241,E2 -5858.241} C_VEL
LIN {X 0,Y 502.811,Z 908.992,A -85,B 0,C 180,E1 -5859.453,E2 -5859.453} C_VEL
LIN {X 0,Y 503.061,Z 900.54,A -85,B 0,C 180,E1 -5860.464,E2 -5860.464} C_VEL
LIN {X 0,Y 503.539,Z 890.09,A -85,B 0,C 180,E1 -5861.472,E2 -5861.472} C_VEL
LIN {X 0,Y 503.873,Z 879.576,A -85,B 0,C 180,E1 -5862.291,E2 -5862.291} C_VEL
LIN {X 0,Y 504.122,Z 868.24,A -85,B 0,C 180,E1 -5862.991,E2 -5862.991} C_VEL
LIN {X 0,Y 504.473,Z 856.458,A -85,B 0,C 180,E1 -5863.546,E2 -5863.546} C_VEL
LIN {X 0,Y 504.72,Z 843.837,A -85,B 0,C 180,E1 -5863.975,E2 -5863.975} C_VEL
LIN {X 0,Y 503.56,Z 834.82,A -85,B 0,C 180,E1 -5864.224,E2 -5864.224} C_VEL
LIN {X 0,Y 502.827,Z 829.599,A -85,B 0,C 180,E1 -5864.348,E2 -5864.348} C_VEL
LIN {X 0,Y 503.111,Z 814.087,A -85,B 0,C 180,E1 -5867.478,E2 -5867.478} C_VEL
LIN {X 0,Y 503.428,Z 798.119,A -85,B 0,C 180,E1 -5870.717,E2 -5870.717} C_VEL
LIN {X 0,Y 503.767,Z 783.078,A -85,B 0,C 180,E1 -5873.865,E2 -5873.865} C_VEL
LIN {X 0,Y 504.169,Z 769.074,A -85,B 0,C 180,E1 -5876.856,E2 -5876.856} C_VEL
LIN {X 0,Y 504.595,Z 753.519,A -85,B 0,C 180,E1 -5880.284,E2 -5880.284} C_VEL
LIN {X 0,Y 505.076,Z 739.852,A -85,B 0,C 180,E1 -5883.396,E2 -5883.396} C_VEL
LIN {X 0,Y 505.481,Z 727.75,A -85,B 0,C 180,E1 -5886.253,E2 -5886.253} C_VEL
LIN {X 0,Y 504.098,Z 720.133,A -85,B 0,C 180,E1 -5888.218,E2 -5888.218} C_VEL
LIN {X 0,Y 502.816,Z 713.854,A -85,B 0,C 180,E1 -5889.932,E2 -5889.932} C_VEL
LIN {X 0,Y 502.805,Z 713.852,A -85,B 0,C 180,E1 -5892.199,E2 -5892.199} C_VEL
LIN {X 0,Y 502.803,Z 713.856,A -85,B 0,C 180,E1 -5895.468,E2 -5895.468} C_VEL
LIN {X 0,Y 502.823,Z 713.85,A -85,B 0,C 180,E1 -5898.934,E2 -5898.934} C_VEL
LIN {X 0,Y 502.796,Z 713.851,A -85,B 0,C 180,E1 -5902.046,E2 -5902.046} C_VEL
LIN {X 0,Y 502.802,Z 713.852,A -85,B 0,C 180,E1 -5905.034,E2 -5905.034} C_VEL
LIN {X 0,Y 502.787,Z 713.855,A -85,B 0,C 180,E1 -5907.916,E2 -5907.916} C_VEL
LIN {X 0,Y 502.827,Z 713.846,A -85,B 0,C 180,E1 -5910.712,E2 -5910.712} C_VEL
LIN {X 0,Y 502.865,Z 713.846,A -85,B 0,C 180,E1 -5913.439,E2 -5913.439} C_VEL
LIN {X 0,Y 502.778,Z 713.856,A -85,B 0,C 180,E1 -5916.086,E2 -5916.086} C_VEL
LIN {X 0,Y 502.786,Z 713.851,A -85,B 0,C 180,E1 -5918.689,E2 -5918.689} C_VEL
LIN {X 0,Y 502.829,Z 713.848,A -85,B 0,C 180,E1 -5921.248,E2 -5921.248} C_VEL
LIN {X 0,Y 502.852,Z 713.844,A -85,B 0,C 180,E1 -5924.6,E2 -5924.6} C_VEL
LIN {X 0,Y 502.88,Z 713.848,A -85,B 0,C 180,E1 -5928.039,E2 -5928.039} C_VEL
LIN {X 0,Y 502.872,Z 713.841,A -85,B 0,C 180,E1 -5931.157,E2 -5931.157} C_VEL
LIN {X 0,Y 502.913,Z 713.839,A -85,B 0,C 180,E1 -5933.581,E2 -5933.581} C_VEL
LIN {X 0,Y 502.867,Z 713.843,A -85,B 0,C 180,E1 -5936.795,E2 -5936.795} C_VEL
LIN {X 0,Y 502.899,Z 713.843,A -85,B 0,C 180,E1 -5938.398,E2 -5938.398} C_VEL
LIN {X 0,Y 502.993,Z 713.827,A -85,B 0,C 180,E1 -5940.801,E2 -5940.801} C_VEL
LIN {X 0,Y 503.021,Z 713.828,A -85,B 0,C 180,E1 -5942.402,E2 -5942.402} C_VEL
LIN {X 0,Y 502.925,Z 713.836,A -85,B 0,C 180,E1 -5945.614,E2 -5945.614} C_VEL
LIN {X 0,Y 502.87,Z 713.843,A -85,B 0,C 180,E1 -5948.843,E2 -5948.843} C_VEL
LIN {X 0,Y 502.848,Z 713.849,A -85,B 0,C 180,E1 -5952.102,E2 -5952.102} C_VEL
LIN {X 0,Y 502.851,Z 713.844,A -85,B 0,C 180,E1 -5955.4,E2 -5955.4} C_VEL
LIN {X 0,Y 502.825,Z 713.852,A -85,B 0,C 180,E1 -5958.752,E2 -5958.752} C_VEL
LIN {X 0,Y 502.786,Z 713.853,A -85,B 0,C 180,E1 -5961.311,E2 -5961.311} C_VEL
LIN {X 0,Y 502.769,Z 713.856,A -85,B 0,C 180,E1 -5963.915,E2 -5963.915} C_VEL
LIN {X 0,Y 502.784,Z 713.858,A -85,B 0,C 180,E1 -5966.571,E2 -5966.571} C_VEL
LIN {X 0,Y 502.814,Z 713.85,A -85,B 0,C 180,E1 -5969.289,E2 -5969.289} C_VEL
LIN {X 0,Y 502.784,Z 713.854,A -85,B 0,C 180,E1 -5972.085,E2 -5972.085} C_VEL
LIN {X 0,Y 502.793,Z 713.857,A -85,B 0,C 180,E1 -5974.967,E2 -5974.967} C_VEL
LIN {X 0,Y 502.766,Z 713.855,A -85,B 0,C 180,E1 -5977.957,E2 -5977.957} C_VEL
LIN {X 0,Y 502.764,Z 713.861,A -85,B 0,C 180,E1 -5981.072,E2 -5981.072} C_VEL
LIN {X 0,Y 502.787,Z 713.856,A -85,B 0,C 180,E1 -5984.53,E2 -5984.53} C_VEL
LIN {X 0,Y 502.768,Z 713.855,A -85,B 0,C 180,E1 -5987.858,E2 -5987.858} C_VEL
LIN {X 0,Y 502.783,Z 713.858,A -85,B 0,C 180,E1 -5991.022,E2 -5991.022} C_VEL
LIN {X 0,Y 502.754,Z 713.857,A -85,B 0,C 180,E1 -5994.173,E2 -5994.173} C_VEL
LIN {X 0,Y 502.772,Z 713.86,A -85,B 0,C 180,E1 -5997.005,E2 -5997.005} C_VEL
LIN {X 0,Y 502.758,Z 713.859,A -85,B 0,C 180,E1 -5997.203,E2 -5997.203} C_VEL
LIN {X 0,Y 502.075,Z 713.943,A -85,B 0,C 180,E1 -5997.872,E2 -5997.872} C_VEL
LIN {X 0,Y 499.226,Z 714.302,A -85,B 0,C 180,E1 -5998.958,E2 -5998.958} C_VEL
LIN {X 0,Y 496.827,Z 714.597,A -85,B 0,C 180,E1 -5999.833,E2 -5999.833} C_VEL
LIN {X 0,Y 495.798,Z 714.724,A -85,B 0,C 180,E1 -6000.509,E2 -6000.509} C_VEL
LIN {X 0,Y 495.714,Z 714.734,A -85,B 0,C 180,E1 -6000.738,E2 -6000.738} C_VEL
LIN {X 0,Y 495.706,Z 714.735,A -85,B 0,C 180,E1 -6003.927,E2 -6003.927} C_VEL
LIN {X 0,Y 495.76,Z 714.733,A -85,B 0,C 180,E1 -6007.14,E2 -6007.14} C_VEL
LIN {X 0,Y 495.77,Z 714.727,A -85,B 0,C 180,E1 -6010.11,E2 -6010.11} C_VEL
LIN {X 0,Y 495.742,Z 714.731,A -85,B 0,C 180,E1 -6012.68,E2 -6012.68} C_VEL
LIN {X 0,Y 495.78,Z 714.731,A -85,B 0,C 180,E1 -6015.217,E2 -6015.217} C_VEL
LIN {X 0,Y 495.823,Z 714.72,A -85,B 0,C 180,E1 -6018.554,E2 -6018.554} C_VEL
LIN {X 0,Y 495.812,Z 714.725,A -85,B 0,C 180,E1 -6021.851,E2 -6021.851} C_VEL
LIN {X 0,Y 495.854,Z 714.717,A -85,B 0,C 180,E1 -6024.306,E2 -6024.306} C_VEL
LIN {X 0,Y 495.978,Z 714.707,A -85,B 0,C 180,E1 -6027.564,E2 -6027.564} C_VEL
LIN {X 0,Y 495.975,Z 714.704,A -85,B 0,C 180,E1 -6030,E2 -6030} C_VEL
LIN {X 0,Y 495.979,Z 714.701,A -85,B 0,C 180,E1 -6032.436,E2 -6032.436} C_VEL
LIN {X 0,Y 495.858,Z 714.722,A -85,B 0,C 180,E1 -6035.694,E2 -6035.694} C_VEL
LIN {X 0,Y 495.817,Z 714.724,A -85,B 0,C 180,E1 -6038.149,E2 -6038.149} C_VEL
LIN {X 0,Y 495.855,Z 714.718,A -85,B 0,C 180,E1 -6041.445,E2 -6041.445} C_VEL
LIN {X 0,Y 495.793,Z 714.723,A -85,B 0,C 180,E1 -6044.783,E2 -6044.783} C_VEL
LIN {X 0,Y 495.783,Z 714.729,A -85,B 0,C 180,E1 -6048.172,E2 -6048.172} C_VEL
LIN {X 0,Y 495.779,Z 714.725,A -85,B 0,C 180,E1 -6050.756,E2 -6050.756} C_VEL
LIN {X 0,Y 495.744,Z 714.729,A -85,B 0,C 180,E1 -6053.388,E2 -6053.388} C_VEL
LIN {X 0,Y 495.746,Z 714.73,A -85,B 0,C 180,E1 -6056.731,E2 -6056.731} C_VEL
LIN {X 0,Y 495.766,Z 714.728,A -85,B 0,C 180,E1 -6059.747,E2 -6059.747} C_VEL
LIN {X 0,Y 495.77,Z 714.729,A -85,B 0,C 180,E1 -6062.594,E2 -6062.594} C_VEL
LIN {X 0,Y 495.751,Z 714.728,A -85,B 0,C 180,E1 -6065.538,E2 -6065.538} C_VEL
LIN {X 0,Y 495.767,Z 714.728,A -85,B 0,C 180,E1 -6068.768,E2 -6068.768} C_VEL
LIN {X 0,Y 495.76,Z 714.727,A -85,B 0,C 180,E1 -6071.781,E2 -6071.781} C_VEL
LIN {X 0,Y 495.741,Z 714.73,A -85,B 0,C 180,E1 -6075.141,E2 -6075.141} C_VEL
LIN {X 0,Y 495.784,Z 714.731,A -85,B 0,C 180,E1 -6078.332,E2 -6078.332} C_VEL
LIN {X 0,Y 497.714,Z 721.801,A -85,B 0,C 180,E1 -6078.74,E2 -6078.74} C_VEL
LIN {X 0,Y 497.441,Z 734.025,A -85,B 0,C 180,E1 -6079.465,E2 -6079.465} C_VEL
LIN {X 0,Y 497.109,Z 744.306,A -85,B 0,C 180,E1 -6080.239,E2 -6080.239} C_VEL
LIN {X 0,Y 496.844,Z 753.368,A -85,B 0,C 180,E1 -6081.078,E2 -6081.078} C_VEL
LIN {X 0,Y 496.559,Z 762.041,A -85,B 0,C 180,E1 -6082.05,E2 -6082.05} C_VEL
LIN {X 0,Y 496.187,Z 770.721,A -85,B 0,C 180,E1 -6083.242,E2 -6083.242} C_VEL
LIN {X 0,Y 495.977,Z 777.979,A -85,B 0,C 180,E1 -6084.481,E2 -6084.481} C_VEL
LIN {X 0,Y 495.71,Z 784.675,A -85,B 0,C 180,E1 -6085.943,E2 -6085.943} C_VEL
LIN {X 0,Y 495.56,Z 789.658,A -85,B 0,C 180,E1 -6087.39,E2 -6087.39} C_VEL
LIN {X 0,Y 495.525,Z 792.129,A -85,B 0,C 180,E1 -6088.347,E2 -6088.347} C_VEL
LIN {X 0,Y 495.388,Z 794.961,A -85,B 0,C 180,E1 -6089.929,E2 -6089.929} C_VEL
LIN {X 0,Y 495.346,Z 796.285,A -85,B 0,C 180,E1 -6091.602,E2 -6091.602} C_VEL
LIN {X 0,Y 495.376,Z 795.939,A -85,B 0,C 180,E1 -6093.355,E2 -6093.355} C_VEL
LIN {X 0,Y 495.468,Z 794.215,A -85,B 0,C 180,E1 -6094.815,E2 -6094.815} C_VEL
LIN {X 0,Y 495.589,Z 791.477,A -85,B 0,C 180,E1 -6096.161,E2 -6096.161} C_VEL
LIN {X 0,Y 495.712,Z 787.597,A -85,B 0,C 180,E1 -6097.493,E2 -6097.493} C_VEL
LIN {X 0,Y 495.922,Z 782.456,A -85,B 0,C 180,E1 -6098.815,E2 -6098.815} C_VEL
LIN {X 0,Y 496.159,Z 775.896,A -85,B 0,C 180,E1 -6100.126,E2 -6100.126} C_VEL
LIN {X 0,Y 496.451,Z 768.379,A -85,B 0,C 180,E1 -6101.317,E2 -6101.317} C_VEL
LIN {X 0,Y 496.805,Z 759.088,A -85,B 0,C 180,E1 -6102.506,E2 -6102.506} C_VEL
LIN {X 0,Y 497.132,Z 749.706,A -85,B 0,C 180,E1 -6103.47,E2 -6103.47} C_VEL
LIN {X 0,Y 497.448,Z 739.435,A -85,B 0,C 180,E1 -6104.324,E2 -6104.324} C_VEL
LIN {X 0,Y 497.71,Z 728.26,A -85,B 0,C 180,E1 -6105.066,E2 -6105.066} C_VEL
LIN {X 0,Y 497.822,Z 722.499,A -85,B 0,C 180,E1 -6105.383,E2 -6105.383} C_VEL
LIN {X 0,Y 495.777,Z 714.731,A -85,B 0,C 180,E1 -6105.82,E2 -6105.82} C_VEL
LIN {X 0,Y 495.853,Z 714.719,A -85,B 0,C 180,E1 -6108.555,E2 -6108.555} C_VEL
LIN {X 0,Y 495.841,Z 714.722,A -85,B 0,C 180,E1 -6111.851,E2 -6111.851} C_VEL
LIN {X 0,Y 495.837,Z 714.718,A -85,B 0,C 180,E1 -6115.121,E2 -6115.121} C_VEL
LIN {X 0,Y 495.991,Z 714.705,A -85,B 0,C 180,E1 -6117.564,E2 -6117.564} C_VEL
LIN {X 0,Y 495.966,Z 714.701,A -85,B 0,C 180,E1 -6120.812,E2 -6120.812} C_VEL
LIN {X 0,Y 495.992,Z 714.697,A -85,B 0,C 180,E1 -6122.436,E2 -6122.436} C_VEL
LIN {X 0,Y 495.894,Z 714.715,A -85,B 0,C 180,E1 -6125.693,E2 -6125.693} C_VEL
LIN {X 0,Y 495.84,Z 714.72,A -85,B 0,C 180,E1 -6128.148,E2 -6128.148} C_VEL
LIN {X 0,Y 495.856,Z 714.716,A -85,B 0,C 180,E1 -6131.445,E2 -6131.445} C_VEL
LIN {X 0,Y 495.794,Z 714.72,A -85,B 0,C 180,E1 -6134.783,E2 -6134.783} C_VEL
LIN {X 0,Y 495.775,Z 714.725,A -85,B 0,C 180,E1 -6137.319,E2 -6137.319} C_VEL
LIN {X 0,Y 495.775,Z 714.729,A -85,B 0,C 180,E1 -6139.89,E2 -6139.89} C_VEL
LIN {X 0,Y 495.763,Z 714.727,A -85,B 0,C 180,E1 -6142.86,E2 -6142.86} C_VEL
LIN {X 0,Y 495.785,Z 714.729,A -85,B 0,C 180,E1 -6146.068,E2 -6146.068} C_VEL
LIN {X 0,Y 495.776,Z 714.727,A -85,B 0,C 180,E1 -6148.815,E2 -6148.815} C_VEL
LIN {X 0,Y 495.76,Z 714.727,A -85,B 0,C 180,E1 -6151.725,E2 -6151.725} C_VEL
LIN {X 0,Y 495.773,Z 714.731,A -85,B 0,C 180,E1 -6154.694,E2 -6154.694} C_VEL
LIN {X 0,Y 495.733,Z 714.733,A -85,B 0,C 180,E1 -6157.561,E2 -6157.561} C_VEL
LIN {X 0,Y 495.77,Z 714.735,A -85,B 0,C 180,E1 -6160.7,E2 -6160.7} C_VEL
LIN {X 0,Y 495.738,Z 714.733,A -85,B 0,C 180,E1 -6164.001,E2 -6164.001} C_VEL
LIN {X 0,Y 495.729,Z 714.738,A -85,B 0,C 180,E1 -6167.117,E2 -6167.117} C_VEL
LIN {X 0,Y 495.762,Z 714.737,A -85,B 0,C 180,E1 -6169.953,E2 -6169.953} C_VEL
LIN {X 0,Y 495.793,Z 714.84,A -85,B 0,C 180,E1 -6170.702,E2 -6170.702} C_VEL
LIN {X 0,Y 497.553,Z 723.759,A -85,B 0,C 180,E1 -6173.108,E2 -6173.108} C_VEL
LIN {X 0,Y 497.864,Z 727.911,A -85,B 0,C 180,E1 -6174.138,E2 -6174.138} C_VEL
LIN {X 0,Y 497.536,Z 740.33,A -85,B 0,C 180,E1 -6177.055,E2 -6177.055} C_VEL
LIN {X 0,Y 497.158,Z 753.288,A -85,B 0,C 180,E1 -6179.954,E2 -6179.954} C_VEL
LIN {X 0,Y 496.881,Z 767.821,A -85,B 0,C 180,E1 -6183.088,E2 -6183.088} C_VEL
LIN {X 0,Y 496.596,Z 782.702,A -85,B 0,C 180,E1 -6186.213,E2 -6186.213} C_VEL
LIN {X 0,Y 496.298,Z 797.63,A -85,B 0,C 180,E1 -6189.266,E2 -6189.266} C_VEL
LIN {X 0,Y 496.017,Z 814.665,A -85,B 0,C 180,E1 -6192.69,E2 -6192.69} C_VEL
LIN {X 0,Y 495.722,Z 828.389,A -85,B 0,C 180,E1 -6195.451,E2 -6195.451} C_VEL
LIN {X 0,Y 497.514,Z 841.543,A -85,B 0,C 180,E1 -6195.792,E2 -6195.792} C_VEL
LIN {X 0,Y 497.737,Z 847.533,A -85,B 0,C 180,E1 -6195.981,E2 -6195.981} C_VEL
LIN {X 0,Y 497.315,Z 860.968,A -85,B 0,C 180,E1 -6196.516,E2 -6196.516} C_VEL
LIN {X 0,Y 496.982,Z 873.055,A -85,B 0,C 180,E1 -6197.178,E2 -6197.178} C_VEL
LIN {X 0,Y 496.615,Z 885.455,A -85,B 0,C 180,E1 -6198.055,E2 -6198.055} C_VEL
LIN {X 0,Y 496.207,Z 895.863,A -85,B 0,C 180,E1 -6198.977,E2 -6198.977} C_VEL
LIN {X 0,Y 495.898,Z 905.249,A -85,B 0,C 180,E1 -6200.002,E2 -6200.002} C_VEL
LIN {X 0,Y 495.572,Z 914.398,A -85,B 0,C 180,E1 -6201.231,E2 -6201.231} C_VEL
LIN {X 0,Y 495.316,Z 921.741,A -85,B 0,C 180,E1 -6202.458,E2 -6202.458} C_VEL
LIN {X 0,Y 495.185,Z 927.609,A -85,B 0,C 180,E1 -6203.703,E2 -6203.703} C_VEL
LIN {X 0,Y 495.123,Z 931.372,A -85,B 0,C 180,E1 -6204.706,E2 -6204.706} C_VEL
LIN {X 0,Y 495.049,Z 934.957,A -85,B 0,C 180,E1 -6205.929,E2 -6205.929} C_VEL
LIN {X 0,Y 495.043,Z 936.806,A -85,B 0,C 180,E1 -6206.744,E2 -6206.744} C_VEL
LIN {X 0,Y 494.961,Z 939.181,A -85,B 0,C 180,E1 -6208.373,E2 -6208.373} C_VEL
LIN {X 0,Y 494.898,Z 940,A -85,B 0,C 180,E1 -6210,E2 -6210} C_VEL
LIN {X 0,Y 494.961,Z 939.183,A -85,B 0,C 180,E1 -6211.627,E2 -6211.627} C_VEL
LIN {X 0,Y 495.043,Z 936.81,A -85,B 0,C 180,E1 -6213.255,E2 -6213.255} C_VEL
LIN {X 0,Y 495.029,Z 933.895,A -85,B 0,C 180,E1 -6214.478,E2 -6214.478} C_VEL
LIN {X 0,Y 495.178,Z 929.944,A -85,B 0,C 180,E1 -6215.702,E2 -6215.702} C_VEL
LIN {X 0,Y 495.251,Z 923.908,A -85,B 0,C 180,E1 -6217.112,E2 -6217.112} C_VEL
LIN {X 0,Y 495.485,Z 917.024,A -85,B 0,C 180,E1 -6218.36,E2 -6218.36} C_VEL
LIN {X 0,Y 495.77,Z 908.575,A -85,B 0,C 180,E1 -6219.588,E2 -6219.588} C_VEL
LIN {X 0,Y 496.037,Z 899.92,A -85,B 0,C 180,E1 -6220.614,E2 -6220.614} C_VEL
LIN {X 0,Y 496.489,Z 889.27,A -85,B 0,C 180,E1 -6221.637,E2 -6221.637} C_VEL
LIN {X 0,Y 496.848,Z 878.599,A -85,B 0,C 180,E1 -6222.468,E2 -6222.468} C_VEL
LIN {X 0,Y 497.153,Z 867.234,A -85,B 0,C 180,E1 -6223.176,E2 -6223.176} C_VEL
LIN {X 0,Y 497.529,Z 855.442,A -85,B 0,C 180,E1 -6223.738,E2 -6223.738} C_VEL
LIN {X 0,Y 497.734,Z 842.816,A -85,B 0,C 180,E1 -6224.176,E2 -6224.176} C_VEL
LIN {X 0,Y 495.726,Z 828.762,A -85,B 0,C 180,E1 -6224.549,E2 -6224.549} C_VEL
LIN {X 0,Y 496.047,Z 813.309,A -85,B 0,C 180,E1 -6227.735,E2 -6227.735} C_VEL
LIN {X 0,Y 496.377,Z 798.144,A -85,B 0,C 180,E1 -6230.857,E2 -6230.857} C_VEL
LIN {X 0,Y 496.734,Z 783.414,A -85,B 0,C 180,E1 -6234.002,E2 -6234.002} C_VEL
LIN {X 0,Y 497.175,Z 769.36,A -85,B 0,C 180,E1 -6237.056,E2 -6237.056} C_VEL
LIN {X 0,Y 497.561,Z 755.859,A -85,B 0,C 180,E1 -6240.074,E2 -6240.074} C_VEL
LIN {X 0,Y 498.073,Z 742.535,A -85,B 0,C 180,E1 -6243.146,E2 -6243.146} C_VEL
LIN {X 0,Y 498.568,Z 729.303,A -85,B 0,C 180,E1 -6246.303,E2 -6246.303} C_VEL
LIN {X 0,Y 497.401,Z 722.661,A -85,B 0,C 180,E1 -6248.043,E2 -6248.043} C_VEL
LIN {X 0,Y 495.787,Z 714.73,A -85,B 0,C 180,E1 -6250.206,E2 -6250.206} C_VEL
LIN {X 0,Y 495.728,Z 714.737,A -85,B 0,C 180,E1 -6252.883,E2 -6252.883} C_VEL
LIN {X 0,Y 495.737,Z 714.731,A -85,B 0,C 180,E1 -6255.999,E2 -6255.999} C_VEL
LIN {X 0,Y 495.769,Z 714.733,A -85,B 0,C 180,E1 -6259.3,E2 -6259.3} C_VEL
LIN {X 0,Y 495.732,Z 714.73,A -85,B 0,C 180,E1 -6262.438,E2 -6262.438} C_VEL
LIN {X 0,Y 495.781,Z 714.731,A -85,B 0,C 180,E1 -6265.457,E2 -6265.457} C_VEL
LIN {X 0,Y 495.759,Z 714.727,A -85,B 0,C 180,E1 -6268.364,E2 -6268.364} C_VEL
LIN {X 0,Y 495.79,Z 714.729,A -85,B 0,C 180,E1 -6271.507,E2 -6271.507} C_VEL
LIN {X 0,Y 495.783,Z 714.729,A -85,B 0,C 180,E1 -6273.932,E2 -6273.932} C_VEL
LIN {X 0,Y 495.761,Z 714.728,A -85,B 0,C 180,E1 -6277.14,E2 -6277.14} C_VEL
LIN {X 0,Y 495.774,Z 714.729,A -85,B 0,C 180,E1 -6280.11,E2 -6280.11} C_VEL
LIN {X 0,Y 495.768,Z 714.726,A -85,B 0,C 180,E1 -6282.681,E2 -6282.681} C_VEL
LIN {X 0,Y 495.793,Z 714.724,A -85,B 0,C 180,E1 -6285.217,E2 -6285.217} C_VEL
LIN {X 0,Y 495.854,Z 714.717,A -85,B 0,C 180,E1 -6288.555,E2 -6288.555} C_VEL
LIN {X 0,Y 495.875,Z 714.718,A -85,B 0,C 180,E1 -6291.852,E2 -6291.852} C_VEL
LIN {X 0,Y 495.893,Z 714.716,A -85,B 0,C 180,E1 -6294.307,E2 -6294.307} C_VEL
LIN {X 0,Y 495.989,Z 714.701,A -85,B 0,C 180,E1 -6297.564,E2 -6297.564} C_VEL
LIN {X 0,Y 495.945,Z 714.705,A -85,B 0,C 180,E1 -6300.812,E2 -6300.812} C_VEL
LIN {X 0,Y 495.989,Z 714.704,A -85,B 0,C 180,E1 -6302.436,E2 -6302.436} C_VEL
LIN {X 0,Y 495.88,Z 714.715,A -85,B 0,C 180,E1 -6305.694,E2 -6305.694} C_VEL
LIN {X 0,Y 495.839,Z 714.719,A -85,B 0,C 180,E1 -6308.97,E2 -6308.97} C_VEL
LIN {X 0,Y 495.831,Z 714.723,A -85,B 0,C 180,E1 -6312.035,E2 -6312.035} C_VEL
LIN {X 0,Y 495.826,Z 714.719,A -85,B 0,C 180,E1 -6315.451,E2 -6315.451} C_VEL
LIN {X 0,Y 495.781,Z 714.727,A -85,B 0,C 180,E1 -6319.029,E2 -6319.029} C_VEL
LIN {X 0,Y 495.745,Z 714.73,A -85,B 0,C 180,E1 -6321.629,E2 -6321.629} C_VEL
LIN {X 0,Y 495.715,Z 714.738,A -85,B 0,C 180,E1 -6324.277,E2 -6324.277} C_VEL
LIN {X 0,Y 495.733,Z 714.735,A -85,B 0,C 180,E1 -6326.979,E2 -6326.979} C_VEL
LIN {X 0,Y 495.765,Z 714.73,A -85,B 0,C 180,E1 -6330.147,E2 -6330.147} C_VEL
LIN {X 0,Y 495.753,Z 714.731,A -85,B 0,C 180,E1 -6333.237,E2 -6333.237} C_VEL
LIN {X 0,Y 495.71,Z 714.735,A -85,B 0,C 180,E1 -6336.087,E2 -6336.087} C_VEL
LIN {X 0,Y 495.741,Z 714.735,A -85,B 0,C 180,E1 -6338.765,E2 -6338.765} C_VEL
LIN {X 0,Y 495.725,Z 714.732,A -85,B 0,C 180,E1 -6341.785,E2 -6341.785} C_VEL
LIN {X 0,Y 495.739,Z 714.735,A -85,B 0,C 180,E1 -6345.141,E2 -6345.141} C_VEL
LIN {X 0,Y 495.725,Z 714.733,A -85,B 0,C 180,E1 -6348.215,E2 -6348.215} C_VEL
LIN {X 0,Y 495.741,Z 714.735,A -85,B 0,C 180,E1 -6351.236,E2 -6351.236} C_VEL
LIN {X 0,Y 495.731,Z 714.733,A -85,B 0,C 180,E1 -6354.461,E2 -6354.461} C_VEL
LIN {X 0,Y 495.727,Z 714.737,A -85,B 0,C 180,E1 -6357.403,E2 -6357.403} C_VEL
LIN {X 0,Y 495.741,Z 714.73,A -85,B 0,C 180,E1 -6360.252,E2 -6360.252} C_VEL
LIN {X 0,Y 495.714,Z 714.734,A -85,B 0,C 180,E1 -6360.738,E2 -6360.738} C_VEL
LIN {X 0,Y 495.039,Z 714.822,A -85,B 0,C 180,E1 -6361.417,E2 -6361.417} C_VEL
LIN {X 0,Y 492.163,Z 715.178,A -85,B 0,C 180,E1 -6362.519,E2 -6362.519} C_VEL
LIN {X 0,Y 489.745,Z 715.481,A -85,B 0,C 180,E1 -6363.407,E2 -6363.407} C_VEL
LIN {X 0,Y 488.722,Z 715.605,A -85,B 0,C 180,E1 -6364.093,E2 -6364.093} C_VEL
LIN {X 0,Y 488.648,Z 715.614,A -85,B 0,C 180,E1 -6364.325,E2 -6364.325} C_VEL
LIN {X 0,Y 488.723,Z 715.61,A -85,B 0,C 180,E1 -6367.153,E2 -6367.153} C_VEL
LIN {X 0,Y 488.726,Z 715.607,A -85,B 0,C 180,E1 -6369.811,E2 -6369.811} C_VEL
LIN {X 0,Y 488.701,Z 715.607,A -85,B 0,C 180,E1 -6372.422,E2 -6372.422} C_VEL
LIN {X 0,Y 488.756,Z 715.603,A -85,B 0,C 180,E1 -6374.999,E2 -6374.999} C_VEL
LIN {X 0,Y 488.786,Z 715.597,A -85,B 0,C 180,E1 -6378.387,E2 -6378.387} C_VEL
LIN {X 0,Y 488.756,Z 715.604,A -85,B 0,C 180,E1 -6381.733,E2 -6381.733} C_VEL
LIN {X 0,Y 488.814,Z 715.594,A -85,B 0,C 180,E1 -6384.224,E2 -6384.224} C_VEL
LIN {X 0,Y 488.944,Z 715.583,A -85,B 0,C 180,E1 -6387.529,E2 -6387.529} C_VEL
LIN {X 0,Y 488.944,Z 715.58,A -85,B 0,C 180,E1 -6390,E2 -6390} C_VEL
LIN {X 0,Y 488.945,Z 715.577,A -85,B 0,C 180,E1 -6392.472,E2 -6392.472} C_VEL
LIN {X 0,Y 488.818,Z 715.598,A -85,B 0,C 180,E1 -6395.776,E2 -6395.776} C_VEL
LIN {X 0,Y 488.765,Z 715.602,A -85,B 0,C 180,E1 -6398.267,E2 -6398.267} C_VEL
LIN {X 0,Y 488.809,Z 715.598,A -85,B 0,C 180,E1 -6401.613,E2 -6401.613} C_VEL
LIN {X 0,Y 488.765,Z 715.598,A -85,B 0,C 180,E1 -6405,E2 -6405} C_VEL
LIN {X 0,Y 488.75,Z 715.603,A -85,B 0,C 180,E1 -6408.443,E2 -6408.443} C_VEL
LIN {X 0,Y 488.711,Z 715.605,A -85,B 0,C 180,E1 -6411.071,E2 -6411.071} C_VEL
LIN {X 0,Y 488.675,Z 715.613,A -85,B 0,C 180,E1 -6413.747,E2 -6413.747} C_VEL
LIN {X 0,Y 488.705,Z 715.606,A -85,B 0,C 180,E1 -6416.923,E2 -6416.923} C_VEL
LIN {X 0,Y 488.727,Z 715.61,A -85,B 0,C 180,E1 -6420.219,E2 -6420.219} C_VEL
LIN {X 0,Y 488.733,Z 715.602,A -85,B 0,C 180,E1 -6423.483,E2 -6423.483} C_VEL
LIN {X 0,Y 488.686,Z 715.615,A -85,B 0,C 180,E1 -6426.355,E2 -6426.355} C_VEL
LIN {X 0,Y 488.705,Z 715.605,A -85,B 0,C 180,E1 -6429.254,E2 -6429.254} C_VEL
LIN {X 0,Y 488.711,Z 715.604,A -85,B 0,C 180,E1 -6431.6,E2 -6431.6} C_VEL
LIN {X 0,Y 488.705,Z 715.61,A -85,B 0,C 180,E1 -6434.803,E2 -6434.803} C_VEL
LIN {X 0,Y 488.749,Z 715.728,A -85,B 0,C 180,E1 -6438.145,E2 -6438.145} C_VEL
LIN {X 0,Y 490.838,Z 723.224,A -85,B 0,C 180,E1 -6438.586,E2 -6438.586} C_VEL
LIN {X 0,Y 490.575,Z 734.686,A -85,B 0,C 180,E1 -6439.277,E2 -6439.277} C_VEL
LIN {X 0,Y 490.205,Z 745.344,A -85,B 0,C 180,E1 -6440.087,E2 -6440.087} C_VEL
LIN {X 0,Y 489.876,Z 756.115,A -85,B 0,C 180,E1 -6441.122,E2 -6441.122} C_VEL
LIN {X 0,Y 489.546,Z 764.811,A -85,B 0,C 180,E1 -6442.148,E2 -6442.148} C_VEL
LIN {X 0,Y 489.191,Z 772.937,A -85,B 0,C 180,E1 -6443.315,E2 -6443.315} C_VEL
LIN {X 0,Y 488.953,Z 780.325,A -85,B 0,C 180,E1 -6444.652,E2 -6444.652} C_VEL
LIN {X 0,Y 488.711,Z 785.762,A -85,B 0,C 180,E1 -6445.885,E2 -6445.885} C_VEL
LIN {X 0,Y 488.555,Z 790.735,A -85,B 0,C 180,E1 -6447.354,E2 -6447.354} C_VEL
LIN {X 0,Y 488.468,Z 794.22,A -85,B 0,C 180,E1 -6448.804,E2 -6448.804} C_VEL
LIN {X 0,Y 488.388,Z 795.778,A -85,B 0,C 180,E1 -6449.758,E2 -6449.758} C_VEL
LIN {X 0,Y 488.355,Z 796.841,A -85,B 0,C 180,E1 -6450.705,E2 -6450.705} C_VEL
LIN {X 0,Y 488.333,Z 797.333,A -85,B 0,C 180,E1 -6451.645,E2 -6451.645} C_VEL
LIN {X 0,Y 488.344,Z 797.105,A -85,B 0,C 180,E1 -6453.161,E2 -6453.161} C_VEL
LIN {X 0,Y 488.407,Z 795.895,A -85,B 0,C 180,E1 -6454.425,E2 -6454.425} C_VEL
LIN {X 0,Y 488.508,Z 794.451,A -85,B 0,C 180,E1 -6455.341,E2 -6455.341} C_VEL
LIN {X 0,Y 488.602,Z 792.466,A -85,B 0,C 180,E1 -6456.25,E2 -6456.25} C_VEL
LIN {X 0,Y 488.734,Z 788.569,A -85,B 0,C 180,E1 -6457.6,E2 -6457.6} C_VEL
LIN {X 0,Y 488.969,Z 783.405,A -85,B 0,C 180,E1 -6458.941,E2 -6458.941} C_VEL
LIN {X 0,Y 489.227,Z 776.8,A -85,B 0,C 180,E1 -6460.27,E2 -6460.27} C_VEL
LIN {X 0,Y 489.568,Z 768.477,A -85,B 0,C 180,E1 -6461.589,E2 -6461.589} C_VEL
LIN {X 0,Y 489.927,Z 759.912,A -85,B 0,C 180,E1 -6462.683,E2 -6462.683} C_VEL
LIN {X 0,Y 490.273,Z 750.622,A -85,B 0,C 180,E1 -6463.645,E2 -6463.645} C_VEL
LIN {X 0,Y 490.611,Z 740.111,A -85,B 0,C 180,E1 -6464.526,E2 -6464.526} C_VEL
LIN {X 0,Y 490.894,Z 728.844,A -85,B 0,C 180,E1 -6465.278,E2 -6465.278} C_VEL
LIN {X 0,Y 490.88,Z 723.185,A -85,B 0,C 180,E1 -6465.596,E2 -6465.596} C_VEL
LIN {X 0,Y 488.772,Z 715.603,A -85,B 0,C 180,E1 -6466.037,E2 -6466.037} C_VEL
LIN {X 0,Y 488.805,Z 715.598,A -85,B 0,C 180,E1 -6468.387,E2 -6468.387} C_VEL
LIN {X 0,Y 488.79,Z 715.602,A -85,B 0,C 180,E1 -6471.733,E2 -6471.733} C_VEL
LIN {X 0,Y 488.833,Z 715.591,A -85,B 0,C 180,E1 -6474.224,E2 -6474.224} C_VEL
LIN {X 0,Y 488.958,Z 715.581,A -85,B 0,C 180,E1 -6477.529,E2 -6477.529} C_VEL
LIN {X 0,Y 488.918,Z 715.579,A -85,B 0,C 180,E1 -6480.824,E2 -6480.824} C_VEL
LIN {X 0,Y 488.959,Z 715.573,A -85,B 0,C 180,E1 -6482.471,E2 -6482.471} C_VEL
LIN {X 0,Y 488.853,Z 715.592,A -85,B 0,C 180,E1 -6485.776,E2 -6485.776} C_VEL
LIN {X 0,Y 488.789,Z 715.596,A -85,B 0,C 180,E1 -6488.267,E2 -6488.267} C_VEL
LIN {X 0,Y 488.81,Z 715.595,A -85,B 0,C 180,E1 -6491.612,E2 -6491.612} C_VEL
LIN {X 0,Y 488.766,Z 715.595,A -85,B 0,C 180,E1 -6495,E2 -6495} C_VEL
LIN {X 0,Y 488.751,Z 715.605,A -85,B 0,C 180,E1 -6498.442,E2 -6498.442} C_VEL
LIN {X 0,Y 488.711,Z 715.602,A -85,B 0,C 180,E1 -6501.071,E2 -6501.071} C_VEL
LIN {X 0,Y 488.684,Z 715.61,A -85,B 0,C 180,E1 -6503.746,E2 -6503.746} C_VEL
LIN {X 0,Y 488.796,Z 715.596,A -85,B 0,C 180,E1 -6506.943,E2 -6506.943} C_VEL
LIN {X 0,Y 488.714,Z 715.612,A -85,B 0,C 180,E1 -6510.363,E2 -6510.363} C_VEL
LIN {X 0,Y 488.738,Z 715.602,A -85,B 0,C 180,E1 -6513.484,E2 -6513.484} C_VEL
LIN {X 0,Y 488.686,Z 715.616,A -85,B 0,C 180,E1 -6516.354,E2 -6516.354} C_VEL
LIN {X 0,Y 488.705,Z 715.61,A -85,B 0,C 180,E1 -6519.254,E2 -6519.254} C_VEL
LIN {X 0,Y 488.711,Z 715.608,A -85,B 0,C 180,E1 -6521.6,E2 -6521.6} C_VEL
LIN {X 0,Y 488.716,Z 715.612,A -85,B 0,C 180,E1 -6524.801,E2 -6524.801} C_VEL
LIN {X 0,Y 488.695,Z 715.613,A -85,B 0,C 180,E1 -6527.474,E2 -6527.474} C_VEL
LIN {X 0,Y 488.747,Z 715.701,A -85,B 0,C 180,E1 -6530.417,E2 -6530.417} C_VEL
LIN {X 0,Y 490.787,Z 726.246,A -85,B 0,C 180,E1 -6533.313,E2 -6533.313} C_VEL
LIN {X 0,Y 490.793,Z 733.291,A -85,B 0,C 180,E1 -6535.055,E2 -6535.055} C_VEL
LIN {X 0,Y 490.424,Z 744.643,A -85,B 0,C 180,E1 -6537.725,E2 -6537.725} C_VEL
LIN {X 0,Y 490.081,Z 756.224,A -85,B 0,C 180,E1 -6540.347,E2 -6540.347} C_VEL
LIN {X 0,Y 489.802,Z 769.231,A -85,B 0,C 180,E1 -6543.197,E2 -6543.197} C_VEL
LIN {X 0,Y 489.524,Z 783.799,A -85,B 0,C 180,E1 -6546.297,E2 -6546.297} C_VEL
LIN {X 0,Y 489.185,Z 798.839,A -85,B 0,C 180,E1 -6549.427,E2 -6549.427} C_VEL
LIN {X 0,Y 488.924,Z 814.601,A -85,B 0,C 180,E1 -6552.646,E2 -6552.646} C_VEL
LIN {X 0,Y 488.659,Z 827.207,A -85,B 0,C 180,E1 -6555.236,E2 -6555.236} C_VEL
LIN {X 0,Y 489.967,Z 838.324,A -85,B 0,C 180,E1 -6555.515,E2 -6555.515} C_VEL
LIN {X 0,Y 490.792,Z 844.742,A -85,B 0,C 180,E1 -6555.725,E2 -6555.725} C_VEL
LIN {X 0,Y 490.477,Z 857.463,A -85,B 0,C 180,E1 -6556.218,E2 -6556.218} C_VEL
LIN {X 0,Y 490.041,Z 869.231,A -85,B 0,C 180,E1 -6556.832,E2 -6556.832} C_VEL
LIN {X 0,Y 489.703,Z 880.258,A -85,B 0,C 180,E1 -6557.568,E2 -6557.568} C_VEL
LIN {X 0,Y 489.296,Z 891.421,A -85,B 0,C 180,E1 -6558.504,E2 -6558.504} C_VEL
LIN {X 0,Y 488.931,Z 900.528,A -85,B 0,C 180,E1 -6559.439,E2 -6559.439} C_VEL
LIN {X 0,Y 488.613,Z 910.453,A -85,B 0,C 180,E1 -6560.688,E2 -6560.688} C_VEL
LIN {X 0,Y 488.349,Z 918.371,A -85,B 0,C 180,E1 -6561.934,E2 -6561.934} C_VEL
LIN {X 0,Y 488.141,Z 925.669,A -85,B 0,C 180,E1 -6563.386,E2 -6563.386} C_VEL
LIN {X 0,Y 488.06,Z 930.54,A -85,B 0,C 180,E1 -6564.629,E2 -6564.629} C_VEL
LIN {X 0,Y 487.974,Z 934.259,A -85,B 0,C 180,E1 -6565.87,E2 -6565.87} C_VEL
LIN {X 0,Y 487.967,Z 936.185,A -85,B 0,C 180,E1 -6566.697,E2 -6566.697} C_VEL
LIN {X 0,Y 487.917,Z 937.621,A -85,B 0,C 180,E1 -6567.523,E2 -6567.523} C_VEL
LIN {X 0,Y 487.888,Z 938.646,A -85,B 0,C 180,E1 -6568.349,E2 -6568.349} C_VEL
LIN {X 0,Y 487.834,Z 939.266,A -85,B 0,C 180,E1 -6569.174,E2 -6569.174} C_VEL
LIN {X 0,Y 487.819,Z 939.49,A -85,B 0,C 180,E1 -6570,E2 -6570} C_VEL
LIN {X 0,Y 487.834,Z 939.271,A -85,B 0,C 180,E1 -6570.825,E2 -6570.825} C_VEL
LIN {X 0,Y 487.888,Z 938.654,A -85,B 0,C 180,E1 -6571.651,E2 -6571.651} C_VEL
LIN {X 0,Y 487.917,Z 937.634,A -85,B 0,C 180,E1 -6572.477,E2 -6572.477} C_VEL
LIN {X 0,Y 487.967,Z 936.205,A -85,B 0,C 180,E1 -6573.303,E2 -6573.303} C_VEL
LIN {X 0,Y 487.946,Z 933.183,A -85,B 0,C 180,E1 -6574.544,E2 -6574.544} C_VEL
LIN {X 0,Y 488.127,Z 929.122,A -85,B 0,C 180,E1 -6575.784,E2 -6575.784} C_VEL
LIN {X 0,Y 488.183,Z 922.846,A -85,B 0,C 180,E1 -6577.237,E2 -6577.237} C_VEL
LIN {X 0,Y 488.441,Z 916.027,A -85,B 0,C 180,E1 -6578.481,E2 -6578.481} C_VEL
LIN {X 0,Y 488.709,Z 907.575,A -85,B 0,C 180,E1 -6579.728,E2 -6579.728} C_VEL
LIN {X 0,Y 489.013,Z 898.917,A -85,B 0,C 180,E1 -6580.768,E2 -6580.768} C_VEL
LIN {X 0,Y 489.461,Z 888.259,A -85,B 0,C 180,E1 -6581.807,E2 -6581.807} C_VEL
LIN {X 0,Y 489.844,Z 877.226,A -85,B 0,C 180,E1 -6582.675,E2 -6582.675} C_VEL
LIN {X 0,Y 490.199,Z 866.227,A -85,B 0,C 180,E1 -6583.367,E2 -6583.367} C_VEL
LIN {X 0,Y 490.573,Z 854.424,A -85,B 0,C 180,E1 -6583.937,E2 -6583.937} C_VEL
LIN {X 0,Y 490.739,Z 843.175,A -85,B 0,C 180,E1 -6584.342,E2 -6584.342} C_VEL
LIN {X 0,Y 488.891,Z 830.296,A -85,B 0,C 180,E1 -6584.703,E2 -6584.703} C_VEL
LIN {X 0,Y 488.641,Z 827.702,A -85,B 0,C 180,E1 -6584.791,E2 -6584.791} C_VEL
LIN {X 0,Y 489,Z 812.384,A -85,B 0,C 180,E1 -6587.999,E2 -6587.999} C_VEL
LIN {X 0,Y 489.364,Z 796.992,A -85,B 0,C 180,E1 -6591.262,E2 -6591.262} C_VEL
LIN {X 0,Y 489.727,Z 782.697,A -85,B 0,C 180,E1 -6594.367,E2 -6594.367} C_VEL
LIN {X 0,Y 490.164,Z 769.418,A -85,B 0,C 180,E1 -6597.311,E2 -6597.311} C_VEL
LIN {X 0,Y 490.624,Z 755.751,A -85,B 0,C 180,E1 -6600.424,E2 -6600.424} C_VEL
LIN {X 0,Y 491.199,Z 741.944,A -85,B 0,C 180,E1 -6603.671,E2 -6603.671} C_VEL
LIN {X 0,Y 491.664,Z 730.981,A -85,B 0,C 180,E1 -6606.327,E2 -6606.327} C_VEL
LIN {X 0,Y 490.567,Z 724.587,A -85,B 0,C 180,E1 -6608.027,E2 -6608.027} C_VEL
LIN {X 0,Y 488.729,Z 715.609,A -85,B 0,C 180,E1 -6610.52,E2 -6610.52} C_VEL
LIN {X 0,Y 488.689,Z 715.613,A -85,B 0,C 180,E1 -6613.654,E2 -6613.654} C_VEL
LIN {X 0,Y 488.689,Z 715.608,A -85,B 0,C 180,E1 -6616.346,E2 -6616.346} C_VEL
LIN {X 0,Y 488.735,Z 715.606,A -85,B 0,C 180,E1 -6619.677,E2 -6619.677} C_VEL
LIN {X 0,Y 488.682,Z 715.609,A -85,B 0,C 180,E1 -6622.841,E2 -6622.841} C_VEL
LIN {X 0,Y 488.733,Z 715.606,A -85,B 0,C 180,E1 -6625.887,E2 -6625.887} C_VEL
LIN {X 0,Y 488.695,Z 715.607,A -85,B 0,C 180,E1 -6628.82,E2 -6628.82} C_VEL
LIN {X 0,Y 488.747,Z 715.608,A -85,B 0,C 180,E1 -6631.671,E2 -6631.671} C_VEL
LIN {X 0,Y 488.73,Z 715.603,A -85,B 0,C 180,E1 -6634.443,E2 -6634.443} C_VEL
LIN {X 0,Y 488.724,Z 715.605,A -85,B 0,C 180,E1 -6637.153,E2 -6637.153} C_VEL
LIN {X 0,Y 488.728,Z 715.61,A -85,B 0,C 180,E1 -6639.811,E2 -6639.811} C_VEL
LIN {X 0,Y 488.718,Z 715.606,A -85,B 0,C 180,E1 -6642.423,E2 -6642.423} C_VEL
LIN {X 0,Y 488.765,Z 715.599,A -85,B 0,C 180,E1 -6645,E2 -6645} C_VEL
LIN {X 0,Y 488.808,Z 715.596,A -85,B 0,C 180,E1 -6648.388,E2 -6648.388} C_VEL
LIN {X 0,Y 488.819,Z 715.596,A -85,B 0,C 180,E1 -6651.734,E2 -6651.734} C_VEL
LIN {X 0,Y 488.851,Z 715.594,A -85,B 0,C 180,E1 -6654.224,E2 -6654.224} C_VEL
LIN {X 0,Y 488.955,Z 715.577,A -85,B 0,C 180,E1 -6657.529,E2 -6657.529} C_VEL
LIN {X 0,Y 488.973,Z 715.577,A -85,B 0,C 180,E1 -6660,E2 -6660} C_VEL
LIN {X 0,Y 488.956,Z 715.58,A -85,B 0,C 180,E1 -6662.471,E2 -6662.471} C_VEL
LIN {X 0,Y 488.837,Z 715.593,A -85,B 0,C 180,E1 -6665.776,E2 -6665.776} C_VEL
LIN {X 0,Y 488.788,Z 715.601,A -85,B 0,C 180,E1 -6668.267,E2 -6668.267} C_VEL
LIN {X 0,Y 488.808,Z 715.595,A -85,B 0,C 180,E1 -6671.613,E2 -6671.613} C_VEL
LIN {X 0,Y 488.759,Z 715.601,A -85,B 0,C 180,E1 -6675.001,E2 -6675.001} C_VEL
LIN {X 0,Y 488.748,Z 715.606,A -85,B 0,C 180,E1 -6678.443,E2 -6678.443} C_VEL
LIN {X 0,Y 488.71,Z 715.608,A -85,B 0,C 180,E1 -6681.071,E2 -6681.071} C_VEL
LIN {X 0,Y 488.672,Z 715.611,A -85,B 0,C 180,E1 -6683.747,E2 -6683.747} C_VEL
LIN {X 0,Y 488.7,Z 715.612,A -85,B 0,C 180,E1 -6686.922,E2 -6686.922} C_VEL
LIN {X 0,Y 488.724,Z 715.608,A -85,B 0,C 180,E1 -6690.22,E2 -6690.22} C_VEL
LIN {X 0,Y 488.712,Z 715.607,A -85,B 0,C 180,E1 -6693.48,E2 -6693.48} C_VEL
LIN {X 0,Y 488.67,Z 715.615,A -85,B 0,C 180,E1 -6696.352,E2 -6696.352} C_VEL
LIN {X 0,Y 488.688,Z 715.612,A -85,B 0,C 180,E1 -6699.256,E2 -6699.256} C_VEL
LIN {X 0,Y 488.668,Z 715.612,A -85,B 0,C 180,E1 -6701.594,E2 -6701.594} C_VEL
LIN {X 0,Y 488.703,Z 715.611,A -85,B 0,C 180,E1 -6704.803,E2 -6704.803} C_VEL
LIN {X 0,Y 488.652,Z 715.616,A -85,B 0,C 180,E1 -6707.47,E2 -6707.47} C_VEL
LIN {X 0,Y 488.705,Z 715.608,A -85,B 0,C 180,E1 -6709.674,E2 -6709.674} C_VEL
LIN {X 0,Y 488.653,Z 715.618,A -85,B 0,C 180,E1 -6712.839,E2 -6712.839} C_VEL
LIN {X 0,Y 488.711,Z 715.607,A -85,B 0,C 180,E1 -6715.886,E2 -6715.886} C_VEL
LIN {X 0,Y 488.668,Z 715.616,A -85,B 0,C 180,E1 -6718.818,E2 -6718.818} C_VEL
LIN {X 0,Y 488.693,Z 715.611,A -85,B 0,C 180,E1 -6721.668,E2 -6721.668} C_VEL
LIN {X 0,Y 488.648,Z 715.614,A -85,B 0,C 180,E1 -6724.325,E2 -6724.325} C_VEL
LIN {X 0,Y 488.008,Z 715.699,A -85,B 0,C 180,E1 -6725.013,E2 -6725.013} C_VEL
LIN {X 0,Y 485.179,Z 716.052,A -85,B 0,C 180,E1 -6726.131,E2 -6726.131} C_VEL
LIN {X 0,Y 482.768,Z 716.352,A -85,B 0,C 180,E1 -6727.032,E2 -6727.032} C_VEL
LIN {X 0,Y 481.725,Z 716.48,A -85,B 0,C 180,E1 -6727.728,E2 -6727.728} C_VEL
LIN {X 0,Y 481.638,Z 716.488,A -85,B 0,C 180,E1 -6727.964,E2 -6727.964} C_VEL
LIN {X 0,Y 481.703,Z 716.479,A -85,B 0,C 180,E1 -6730.393,E2 -6730.393} C_VEL
LIN {X 0,Y 481.663,Z 716.488,A -85,B 0,C 180,E1 -6733.033,E2 -6733.033} C_VEL
LIN {X 0,Y 481.679,Z 716.485,A -85,B 0,C 180,E1 -6735.638,E2 -6735.638} C_VEL
LIN {X 0,Y 481.737,Z 716.475,A -85,B 0,C 180,E1 -6738.215,E2 -6738.215} C_VEL
LIN {X 0,Y 481.714,Z 716.482,A -85,B 0,C 180,E1 -6741.611,E2 -6741.611} C_VEL
LIN {X 0,Y 481.775,Z 716.472,A -85,B 0,C 180,E1 -6744.139,E2 -6744.139} C_VEL
LIN {X 0,Y 481.909,Z 716.459,A -85,B 0,C 180,E1 -6747.493,E2 -6747.493} C_VEL
LIN {X 0,Y 481.913,Z 716.456,A -85,B 0,C 180,E1 -6750,E2 -6750} C_VEL
LIN {X 0,Y 481.911,Z 716.453,A -85,B 0,C 180,E1 -6752.508,E2 -6752.508} C_VEL
LIN {X 0,Y 481.779,Z 716.474,A -85,B 0,C 180,E1 -6755.861,E2 -6755.861} C_VEL
LIN {X 0,Y 481.724,Z 716.478,A -85,B 0,C 180,E1 -6758.389,E2 -6758.389} C_VEL
LIN {X 0,Y 481.755,Z 716.479,A -85,B 0,C 180,E1 -6761.785,E2 -6761.785} C_VEL
LIN {X 0,Y 481.746,Z 716.474,A -85,B 0,C 180,E1 -6765.224,E2 -6765.224} C_VEL
LIN {X 0,Y 481.711,Z 716.478,A -85,B 0,C 180,E1 -6768.722,E2 -6768.722} C_VEL
LIN {X 0,Y 481.65,Z 716.486,A -85,B 0,C 180,E1 -6771.395,E2 -6771.395} C_VEL
LIN {X 0,Y 481.653,Z 716.491,A -85,B 0,C 180,E1 -6774.115,E2 -6774.115} C_VEL
LIN {X 0,Y 481.68,Z 716.481,A -85,B 0,C 180,E1 -6777.123,E2 -6777.123} C_VEL
LIN {X 0,Y 481.676,Z 716.484,A -85,B 0,C 180,E1 -6779.742,E2 -6779.742} C_VEL
LIN {X 0,Y 481.674,Z 716.484,A -85,B 0,C 180,E1 -6782.674,E2 -6782.674} C_VEL
LIN {X 0,Y 481.64,Z 716.487,A -85,B 0,C 180,E1 -6785.71,E2 -6785.71} C_VEL
LIN {X 0,Y 481.674,Z 716.483,A -85,B 0,C 180,E1 -6788.859,E2 -6788.859} C_VEL
LIN {X 0,Y 481.656,Z 716.485,A -85,B 0,C 180,E1 -6791.913,E2 -6791.913} C_VEL
LIN {X 0,Y 481.659,Z 716.491,A -85,B 0,C 180,E1 -6794.458,E2 -6794.458} C_VEL
LIN {X 0,Y 481.689,Z 716.484,A -85,B 0,C 180,E1 -6797.933,E2 -6797.933} C_VEL
LIN {X 0,Y 483.907,Z 724.443,A -85,B 0,C 180,E1 -6798.414,E2 -6798.414} C_VEL
LIN {X 0,Y 483.678,Z 736.561,A -85,B 0,C 180,E1 -6799.166,E2 -6799.166} C_VEL
LIN {X 0,Y 483.315,Z 746.578,A -85,B 0,C 180,E1 -6799.95,E2 -6799.95} C_VEL
LIN {X 0,Y 482.969,Z 757.275,A -85,B 0,C 180,E1 -6800.997,E2 -6800.997} C_VEL
LIN {X 0,Y 482.601,Z 766.13,A -85,B 0,C 180,E1 -6802.06,E2 -6802.06} C_VEL
LIN {X 0,Y 482.229,Z 774.563,A -85,B 0,C 180,E1 -6803.306,E2 -6803.306} C_VEL
LIN {X 0,Y 481.98,Z 781.436,A -85,B 0,C 180,E1 -6804.58,E2 -6804.58} C_VEL
LIN {X 0,Y 481.711,Z 786.844,A -85,B 0,C 180,E1 -6805.827,E2 -6805.827} C_VEL
LIN {X 0,Y 481.545,Z 791.813,A -85,B 0,C 180,E1 -6807.316,E2 -6807.316} C_VEL
LIN {X 0,Y 481.49,Z 794.26,A -85,B 0,C 180,E1 -6808.3,E2 -6808.3} C_VEL
LIN {X 0,Y 481.386,Z 796.446,A -85,B 0,C 180,E1 -6809.472,E2 -6809.472} C_VEL
LIN {X 0,Y 481.321,Z 798.18,A -85,B 0,C 180,E1 -6811.175,E2 -6811.175} C_VEL
LIN {X 0,Y 481.31,Z 798.455,A -85,B 0,C 180,E1 -6812.143,E2 -6812.143} C_VEL
LIN {X 0,Y 481.319,Z 798.198,A -85,B 0,C 180,E1 -6813.086,E2 -6813.086} C_VEL
LIN {X 0,Y 481.372,Z 797.487,A -85,B 0,C 180,E1 -6814.024,E2 -6814.024} C_VEL
LIN {X 0,Y 481.466,Z 796.229,A -85,B 0,C 180,E1 -6814.956,E2 -6814.956} C_VEL
LIN {X 0,Y 481.622,Z 793.456,A -85,B 0,C 180,E1 -6816.341,E2 -6816.341} C_VEL
LIN {X 0,Y 481.753,Z 789.546,A -85,B 0,C 180,E1 -6817.71,E2 -6817.71} C_VEL
LIN {X 0,Y 481.977,Z 784.881,A -85,B 0,C 180,E1 -6818.944,E2 -6818.944} C_VEL
LIN {X 0,Y 482.271,Z 778.924,A -85,B 0,C 180,E1 -6820.195,E2 -6820.195} C_VEL
LIN {X 0,Y 482.569,Z 772.351,A -85,B 0,C 180,E1 -6821.313,E2 -6821.313} C_VEL
LIN {X 0,Y 482.919,Z 764.369,A -85,B 0,C 180,E1 -6822.423,E2 -6822.423} C_VEL
LIN {X 0,Y 483.301,Z 755.218,A -85,B 0,C 180,E1 -6823.46,E2 -6823.46} C_VEL
LIN {X 0,Y 483.657,Z 744.957,A -85,B 0,C 180,E1 -6824.406,E2 -6824.406} C_VEL
LIN {X 0,Y 483.94,Z 734.688,A -85,B 0,C 180,E1 -6825.169,E2 -6825.169} C_VEL
LIN {X 0,Y 484.18,Z 725.557,A -85,B 0,C 180,E1 -6825.714,E2 -6825.714} C_VEL
LIN {X 0,Y 481.713,Z 716.481,A -85,B 0,C 180,E1 -6826.259,E2 -6826.259} C_VEL
LIN {X 0,Y 481.707,Z 716.484,A -85,B 0,C 180,E1 -6829.066,E2 -6829.066} C_VEL
LIN {X 0,Y 481.745,Z 716.481,A -85,B 0,C 180,E1 -6831.611,E2 -6831.611} C_VEL
LIN {X 0,Y 481.792,Z 716.469,A -85,B 0,C 180,E1 -6834.139,E2 -6834.139} C_VEL
LIN {X 0,Y 481.924,Z 716.457,A -85,B 0,C 180,E1 -6837.492,E2 -6837.492} C_VEL
LIN {X 0,Y 481.944,Z 716.453,A -85,B 0,C 180,E1 -6840,E2 -6840} C_VEL
LIN {X 0,Y 481.925,Z 716.449,A -85,B 0,C 180,E1 -6842.507,E2 -6842.507} C_VEL
LIN {X 0,Y 481.814,Z 716.468,A -85,B 0,C 180,E1 -6845.86,E2 -6845.86} C_VEL
LIN {X 0,Y 481.744,Z 716.472,A -85,B 0,C 180,E1 -6848.389,E2 -6848.389} C_VEL
LIN {X 0,Y 481.755,Z 716.476,A -85,B 0,C 180,E1 -6851.785,E2 -6851.785} C_VEL
LIN {X 0,Y 481.747,Z 716.469,A -85,B 0,C 180,E1 -6855.224,E2 -6855.224} C_VEL
LIN {X 0,Y 481.712,Z 716.479,A -85,B 0,C 180,E1 -6858.722,E2 -6858.722} C_VEL
LIN {X 0,Y 481.649,Z 716.482,A -85,B 0,C 180,E1 -6861.395,E2 -6861.395} C_VEL
LIN {X 0,Y 481.665,Z 716.486,A -85,B 0,C 180,E1 -6864.114,E2 -6864.114} C_VEL
LIN {X 0,Y 481.75,Z 716.473,A -85,B 0,C 180,E1 -6867.139,E2 -6867.139} C_VEL
LIN {X 0,Y 481.683,Z 716.482,A -85,B 0,C 180,E1 -6869.741,E2 -6869.741} C_VEL
LIN {X 0,Y 481.676,Z 716.486,A -85,B 0,C 180,E1 -6872.674,E2 -6872.674} C_VEL
LIN {X 0,Y 481.64,Z 716.488,A -85,B 0,C 180,E1 -6875.709,E2 -6875.709} C_VEL
LIN {X 0,Y 481.675,Z 716.49,A -85,B 0,C 180,E1 -6878.859,E2 -6878.859} C_VEL
LIN {X 0,Y 481.656,Z 716.488,A -85,B 0,C 180,E1 -6881.913,E2 -6881.913} C_VEL
LIN {X 0,Y 481.663,Z 716.49,A -85,B 0,C 180,E1 -6884.457,E2 -6884.457} C_VEL
LIN {X 0,Y 481.651,Z 716.491,A -85,B 0,C 180,E1 -6887.839,E2 -6887.839} C_VEL
LIN {X 0,Y 481.705,Z 716.604,A -85,B 0,C 180,E1 -6890.14,E2 -6890.14} C_VEL
LIN {X 0,Y 483.738,Z 726.908,A -85,B 0,C 180,E1 -6893.041,E2 -6893.041} C_VEL
LIN {X 0,Y 483.988,Z 730.504,A -85,B 0,C 180,E1 -6893.978,E2 -6893.978} C_VEL
LIN {X 0,Y 483.559,Z 742.782,A -85,B 0,C 180,E1 -6896.974,E2 -6896.974} C_VEL
LIN {X 0,Y 483.159,Z 754.24,A -85,B 0,C 180,E1 -6899.637,E2 -6899.637} C_VEL
LIN {X 0,Y 482.802,Z 768.74,A -85,B 0,C 180,E1 -6902.89,E2 -6902.89} C_VEL
LIN {X 0,Y 482.487,Z 782.737,A -85,B 0,C 180,E1 -6905.93,E2 -6905.93} C_VEL
LIN {X 0,Y 482.128,Z 798.14,A -85,B 0,C 180,E1 -6909.202,E2 -6909.202} C_VEL
LIN {X 0,Y 481.859,Z 813.401,A -85,B 0,C 180,E1 -6912.383,E2 -6912.383} C_VEL
LIN {X 0,Y 481.582,Z 826.022,A -85,B 0,C 180,E1 -6915.014,E2 -6915.014} C_VEL
LIN {X 0,Y 482.908,Z 838.341,A -85,B 0,C 180,E1 -6915.336,E2 -6915.336} C_VEL
LIN {X 0,Y 483.799,Z 845.795,A -85,B 0,C 180,E1 -6915.595,E2 -6915.595} C_VEL
LIN {X 0,Y 483.467,Z 858.491,A -85,B 0,C 180,E1 -6916.122,E2 -6916.122} C_VEL
LIN {X 0,Y 482.971,Z 870.198,A -85,B 0,C 180,E1 -6916.772,E2 -6916.772} C_VEL
LIN {X 0,Y 482.574,Z 881.723,A -85,B 0,C 180,E1 -6917.595,E2 -6917.595} C_VEL
LIN {X 0,Y 482.181,Z 892.424,A -85,B 0,C 180,E1 -6918.545,E2 -6918.545} C_VEL
LIN {X 0,Y 481.819,Z 901.194,A -85,B 0,C 180,E1 -6919.494,E2 -6919.494} C_VEL
LIN {X 0,Y 481.555,Z 909.315,A -85,B 0,C 180,E1 -6920.55,E2 -6920.55} C_VEL
LIN {X 0,Y 481.315,Z 917.262,A -85,B 0,C 180,E1 -6921.815,E2 -6921.815} C_VEL
LIN {X 0,Y 481.081,Z 924.578,A -85,B 0,C 180,E1 -6923.288,E2 -6923.288} C_VEL
LIN {X 0,Y 481.031,Z 929.474,A -85,B 0,C 180,E1 -6924.55,E2 -6924.55} C_VEL
LIN {X 0,Y 480.922,Z 933.204,A -85,B 0,C 180,E1 -6925.81,E2 -6925.81} C_VEL
LIN {X 0,Y 480.925,Z 935.145,A -85,B 0,C 180,E1 -6926.649,E2 -6926.649} C_VEL
LIN {X 0,Y 480.881,Z 936.59,A -85,B 0,C 180,E1 -6927.487,E2 -6927.487} C_VEL
LIN {X 0,Y 480.857,Z 937.622,A -85,B 0,C 180,E1 -6928.325,E2 -6928.325} C_VEL
LIN {X 0,Y 480.806,Z 938.25,A -85,B 0,C 180,E1 -6929.162,E2 -6929.162} C_VEL
LIN {X 0,Y 480.791,Z 938.483,A -85,B 0,C 180,E1 -6930,E2 -6930} C_VEL
LIN {X 0,Y 480.804,Z 938.267,A -85,B 0,C 180,E1 -6930.837,E2 -6930.837} C_VEL
LIN {X 0,Y 480.854,Z 937.654,A -85,B 0,C 180,E1 -6931.675,E2 -6931.675} C_VEL
LIN {X 0,Y 480.877,Z 936.636,A -85,B 0,C 180,E1 -6932.513,E2 -6932.513} C_VEL
LIN {X 0,Y 480.925,Z 935.211,A -85,B 0,C 180,E1 -6933.351,E2 -6933.351} C_VEL
LIN {X 0,Y 480.905,Z 932.192,A -85,B 0,C 180,E1 -6934.61,E2 -6934.61} C_VEL
LIN {X 0,Y 481.067,Z 928.129,A -85,B 0,C 180,E1 -6935.87,E2 -6935.87} C_VEL
LIN {X 0,Y 481.15,Z 921.854,A -85,B 0,C 180,E1 -6937.343,E2 -6937.343} C_VEL
LIN {X 0,Y 481.377,Z 915.027,A -85,B 0,C 180,E1 -6938.606,E2 -6938.606} C_VEL
LIN {X 0,Y 481.657,Z 906.575,A -85,B 0,C 180,E1 -6939.872,E2 -6939.872} C_VEL
LIN {X 0,Y 481.987,Z 897.913,A -85,B 0,C 180,E1 -6940.927,E2 -6940.927} C_VEL
LIN {X 0,Y 482.461,Z 887.25,A -85,B 0,C 180,E1 -6941.981,E2 -6941.981} C_VEL
LIN {X 0,Y 482.864,Z 876.013,A -85,B 0,C 180,E1 -6942.877,E2 -6942.877} C_VEL
LIN {X 0,Y 483.217,Z 865.216,A -85,B 0,C 180,E1 -6943.564,E2 -6943.564} C_VEL
LIN {X 0,Y 483.663,Z 853.412,A -85,B 0,C 180,E1 -6944.14,E2 -6944.14} C_VEL
LIN {X 0,Y 483.714,Z 843.494,A -85,B 0,C 180,E1 -6944.515,E2 -6944.515} C_VEL
LIN {X 0,Y 481.982,Z 830.804,A -85,B 0,C 180,E1 -6944.892,E2 -6944.892} C_VEL
LIN {X 0,Y 481.583,Z 826.9,A -85,B 0,C 180,E1 -6944.986,E2 -6944.986} C_VEL
LIN {X 0,Y 481.958,Z 811.816,A -85,B 0,C 180,E1 -6948.208,E2 -6948.208} C_VEL
LIN {X 0,Y 482.306,Z 796.218,A -85,B 0,C 180,E1 -6951.588,E2 -6951.588} C_VEL
LIN {X 0,Y 482.657,Z 783.986,A -85,B 0,C 180,E1 -6954.29,E2 -6954.29} C_VEL
LIN {X 0,Y 483.13,Z 771.352,A -85,B 0,C 180,E1 -6957.135,E2 -6957.135} C_VEL
LIN {X 0,Y 483.648,Z 756.523,A -85,B 0,C 180,E1 -6960.57,E2 -6960.57} C_VEL
LIN {X 0,Y 484.289,Z 742.844,A -85,B 0,C 180,E1 -6963.835,E2 -6963.835} C_VEL
LIN {X 0,Y 484.733,Z 732.189,A -85,B 0,C 180,E1 -6966.473,E2 -6966.473} C_VEL
LIN {X 0,Y 483.206,Z 723.92,A -85,B 0,C 180,E1 -6968.713,E2 -6968.713} C_VEL
LIN {X 0,Y 481.712,Z 716.484,A -85,B 0,C 180,E1 -6970.865,E2 -6970.865} C_VEL
LIN {X 0,Y 481.662,Z 716.485,A -85,B 0,C 180,E1 -6974.457,E2 -6974.457} C_VEL
LIN {X 0,Y 481.65,Z 716.488,A -85,B 0,C 180,E1 -6977.839,E2 -6977.839} C_VEL
LIN {X 0,Y 481.683,Z 716.48,A -85,B 0,C 180,E1 -6980.651,E2 -6980.651} C_VEL
LIN {X 0,Y 481.63,Z 716.493,A -85,B 0,C 180,E1 -6983.376,E2 -6983.376} C_VEL
LIN {X 0,Y 481.712,Z 716.477,A -85,B 0,C 180,E1 -6986.33,E2 -6986.33} C_VEL
LIN {X 0,Y 481.653,Z 716.489,A -85,B 0,C 180,E1 -6989.417,E2 -6989.417} C_VEL
LIN {X 0,Y 481.702,Z 716.48,A -85,B 0,C 180,E1 -6992.168,E2 -6992.168} C_VEL
LIN {X 0,Y 481.695,Z 716.48,A -85,B 0,C 180,E1 -6994.969,E2 -6994.969} C_VEL
LIN {X 0,Y 481.652,Z 716.49,A -85,B 0,C 180,E1 -6997.705,E2 -6997.705} C_VEL
LIN {X 0,Y 481.707,Z 716.479,A -85,B 0,C 180,E1 -7000.393,E2 -7000.393} C_VEL
LIN {X 0,Y 481.682,Z 716.481,A -85,B 0,C 180,E1 -7003.034,E2 -7003.034} C_VEL
LIN {X 0,Y 481.692,Z 716.483,A -85,B 0,C 180,E1 -7005.639,E2 -7005.639} C_VEL
LIN {X 0,Y 481.754,Z 716.477,A -85,B 0,C 180,E1 -7008.215,E2 -7008.215} C_VEL
LIN {X 0,Y 481.764,Z 716.474,A -85,B 0,C 180,E1 -7011.612,E2 -7011.612} C_VEL
LIN {X 0,Y 481.812,Z 716.472,A -85,B 0,C 180,E1 -7014.14,E2 -7014.14} C_VEL
LIN {X 0,Y 481.921,Z 716.453,A -85,B 0,C 180,E1 -7017.493,E2 -7017.493} C_VEL
LIN {X 0,Y 481.943,Z 716.453,A -85,B 0,C 180,E1 -7020,E2 -7020} C_VEL
LIN {X 0,Y 481.922,Z 716.456,A -85,B 0,C 180,E1 -7022.508,E2 -7022.508} C_VEL
LIN {X 0,Y 481.796,Z 716.47,A -85,B 0,C 180,E1 -7025.861,E2 -7025.861} C_VEL
LIN {X 0,Y 481.743,Z 716.479,A -85,B 0,C 180,E1 -7028.389,E2 -7028.389} C_VEL
LIN {X 0,Y 481.754,Z 716.475,A -85,B 0,C 180,E1 -7031.785,E2 -7031.785} C_VEL
LIN {X 0,Y 481.742,Z 716.474,A -85,B 0,C 180,E1 -7035.224,E2 -7035.224} C_VEL
LIN {X 0,Y 481.71,Z 716.483,A -85,B 0,C 180,E1 -7038.722,E2 -7038.722} C_VEL
LIN {X 0,Y 481.648,Z 716.486,A -85,B 0,C 180,E1 -7041.395,E2 -7041.395} C_VEL
LIN {X 0,Y 481.65,Z 716.489,A -85,B 0,C 180,E1 -7044.115,E2 -7044.115} C_VEL
LIN {X 0,Y 481.675,Z 716.485,A -85,B 0,C 180,E1 -7047.122,E2 -7047.122} C_VEL
LIN {X 0,Y 481.674,Z 716.483,A -85,B 0,C 180,E1 -7049.742,E2 -7049.742} C_VEL
LIN {X 0,Y 481.654,Z 716.489,A -85,B 0,C 180,E1 -7052.676,E2 -7052.676} C_VEL
LIN {X 0,Y 481.63,Z 716.488,A -85,B 0,C 180,E1 -7055.71,E2 -7055.71} C_VEL
LIN {X 0,Y 481.633,Z 716.492,A -85,B 0,C 180,E1 -7058.863,E2 -7058.863} C_VEL
LIN {X 0,Y 481.622,Z 716.489,A -85,B 0,C 180,E1 -7061.909,E2 -7061.909} C_VEL
LIN {X 0,Y 481.656,Z 716.488,A -85,B 0,C 180,E1 -7064.458,E2 -7064.458} C_VEL
LIN {X 0,Y 481.617,Z 716.494,A -85,B 0,C 180,E1 -7066.855,E2 -7066.855} C_VEL
LIN {X 0,Y 481.657,Z 716.485,A -85,B 0,C 180,E1 -7070.057,E2 -7070.057} C_VEL
LIN {X 0,Y 481.61,Z 716.495,A -85,B 0,C 180,E1 -7073.38,E2 -7073.38} C_VEL
LIN {X 0,Y 481.673,Z 716.484,A -85,B 0,C 180,E1 -7076.327,E2 -7076.327} C_VEL
LIN {X 0,Y 481.629,Z 716.492,A -85,B 0,C 180,E1 -7079.422,E2 -7079.422} C_VEL
LIN {X 0,Y 481.647,Z 716.486,A -85,B 0,C 180,E1 -7082.165,E2 -7082.165} C_VEL
LIN {X 0,Y 481.667,Z 716.488,A -85,B 0,C 180,E1 -7084.967,E2 -7084.967} C_VEL
LIN {X 0,Y 481.638,Z 716.488,A -85,B 0,C 180,E1 -7087.964,E2 -7087.964} C_VEL
LIN {X 0,Y 480.971,Z 716.573,A -85,B 0,C 180,E1 -7088.662,E2 -7088.662} C_VEL
LIN {X 0,Y 478.148,Z 716.925,A -85,B 0,C 180,E1 -7089.796,E2 -7089.796} C_VEL
LIN {X 0,Y 475.761,Z 717.223,A -85,B 0,C 180,E1 -7090.71,E2 -7090.71} C_VEL
LIN {X 0,Y 474.732,Z 717.351,A -85,B 0,C 180,E1 -7091.416,E2 -7091.416} C_VEL
LIN {X 0,Y 474.646,Z 717.361,A -85,B 0,C 180,E1 -7091.655,E2 -7091.655} C_VEL
LIN {X 0,Y 474.7,Z 717.352,A -85,B 0,C 180,E1 -7094.544,E2 -7094.544} C_VEL
LIN {X 0,Y 474.695,Z 717.354,A -85,B 0,C 180,E1 -7098.037,E2 -7098.037} C_VEL
LIN {X 0,Y 474.663,Z 717.361,A -85,B 0,C 180,E1 -7101.485,E2 -7101.485} C_VEL
LIN {X 0,Y 474.739,Z 717.349,A -85,B 0,C 180,E1 -7104.052,E2 -7104.052} C_VEL
LIN {X 0,Y 474.874,Z 717.336,A -85,B 0,C 180,E1 -7107.455,E2 -7107.455} C_VEL
LIN {X 0,Y 474.883,Z 717.331,A -85,B 0,C 180,E1 -7110,E2 -7110} C_VEL
LIN {X 0,Y 474.876,Z 717.33,A -85,B 0,C 180,E1 -7112.545,E2 -7112.545} C_VEL
LIN {X 0,Y 474.742,Z 717.349,A -85,B 0,C 180,E1 -7115.948,E2 -7115.948} C_VEL
LIN {X 0,Y 474.7,Z 717.352,A -85,B 0,C 180,E1 -7118.514,E2 -7118.514} C_VEL
LIN {X 0,Y 474.708,Z 717.355,A -85,B 0,C 180,E1 -7121.962,E2 -7121.962} C_VEL
LIN {X 0,Y 474.703,Z 717.353,A -85,B 0,C 180,E1 -7125.456,E2 -7125.456} C_VEL
LIN {X 0,Y 474.666,Z 717.355,A -85,B 0,C 180,E1 -7129.01,E2 -7129.01} C_VEL
LIN {X 0,Y 474.593,Z 717.368,A -85,B 0,C 180,E1 -7131.729,E2 -7131.729} C_VEL
LIN {X 0,Y 474.631,Z 717.362,A -85,B 0,C 180,E1 -7134.495,E2 -7134.495} C_VEL
LIN {X 0,Y 474.64,Z 717.358,A -85,B 0,C 180,E1 -7137.324,E2 -7137.324} C_VEL
LIN {X 0,Y 474.606,Z 717.369,A -85,B 0,C 180,E1 -7140.23,E2 -7140.23} C_VEL
LIN {X 0,Y 474.629,Z 717.359,A -85,B 0,C 180,E1 -7143.221,E2 -7143.221} C_VEL
LIN {X 0,Y 474.593,Z 717.371,A -85,B 0,C 180,E1 -7146.324,E2 -7146.324} C_VEL
LIN {X 0,Y 474.622,Z 717.36,A -85,B 0,C 180,E1 -7149.646,E2 -7149.646} C_VEL
LIN {X 0,Y 474.628,Z 717.365,A -85,B 0,C 180,E1 -7152.237,E2 -7152.237} C_VEL
LIN {X 0,Y 474.621,Z 717.361,A -85,B 0,C 180,E1 -7155.298,E2 -7155.298} C_VEL
LIN {X 0,Y 474.635,Z 717.399,A -85,B 0,C 180,E1 -7157.732,E2 -7157.732} C_VEL
LIN {X 0,Y 477.12,Z 726.856,A -85,B 0,C 180,E1 -7158.309,E2 -7158.309} C_VEL
LIN {X 0,Y 476.815,Z 737.828,A -85,B 0,C 180,E1 -7159.011,E2 -7159.011} C_VEL
LIN {X 0,Y 476.39,Z 748.487,A -85,B 0,C 180,E1 -7159.871,E2 -7159.871} C_VEL
LIN {X 0,Y 476.022,Z 759.496,A -85,B 0,C 180,E1 -7160.984,E2 -7160.984} C_VEL
LIN {X 0,Y 475.587,Z 768.919,A -85,B 0,C 180,E1 -7162.174,E2 -7162.174} C_VEL
LIN {X 0,Y 475.194,Z 777.245,A -85,B 0,C 180,E1 -7163.484,E2 -7163.484} C_VEL
LIN {X 0,Y 474.937,Z 783.718,A -85,B 0,C 180,E1 -7164.752,E2 -7164.752} C_VEL
LIN {X 0,Y 474.701,Z 788.836,A -85,B 0,C 180,E1 -7166.006,E2 -7166.006} C_VEL
LIN {X 0,Y 474.54,Z 792.728,A -85,B 0,C 180,E1 -7167.221,E2 -7167.221} C_VEL
LIN {X 0,Y 474.436,Z 796.339,A -85,B 0,C 180,E1 -7168.77,E2 -7168.77} C_VEL
LIN {X 0,Y 474.349,Z 797.896,A -85,B 0,C 180,E1 -7169.752,E2 -7169.752} C_VEL
LIN {X 0,Y 474.301,Z 799.081,A -85,B 0,C 180,E1 -7170.956,E2 -7170.956} C_VEL
LIN {X 0,Y 474.309,Z 799.44,A -85,B 0,C 180,E1 -7172.655,E2 -7172.655} C_VEL
LIN {X 0,Y 474.32,Z 798.922,A -85,B 0,C 180,E1 -7173.608,E2 -7173.608} C_VEL
LIN {X 0,Y 474.433,Z 797.829,A -85,B 0,C 180,E1 -7174.639,E2 -7174.639} C_VEL
LIN {X 0,Y 474.581,Z 795.523,A -85,B 0,C 180,E1 -7175.968,E2 -7175.968} C_VEL
LIN {X 0,Y 474.745,Z 791.982,A -85,B 0,C 180,E1 -7177.362,E2 -7177.362} C_VEL
LIN {X 0,Y 474.965,Z 787.029,A -85,B 0,C 180,E1 -7178.782,E2 -7178.782} C_VEL
LIN {X 0,Y 475.266,Z 781.009,A -85,B 0,C 180,E1 -7180.116,E2 -7180.116} C_VEL
LIN {X 0,Y 475.676,Z 773.141,A -85,B 0,C 180,E1 -7181.495,E2 -7181.495} C_VEL
LIN {X 0,Y 476.039,Z 765.232,A -85,B 0,C 180,E1 -7182.605,E2 -7182.605} C_VEL
LIN {X 0,Y 476.469,Z 755.389,A -85,B 0,C 180,E1 -7183.725,E2 -7183.725} C_VEL
LIN {X 0,Y 476.862,Z 744.435,A -85,B 0,C 180,E1 -7184.725,E2 -7184.725} C_VEL
LIN {X 0,Y 477.151,Z 733.717,A -85,B 0,C 180,E1 -7185.499,E2 -7185.499} C_VEL
LIN {X 0,Y 477.245,Z 726.375,A -85,B 0,C 180,E1 -7185.937,E2 -7185.937} C_VEL
LIN {X 0,Y 474.665,Z 717.359,A -85,B 0,C 180,E1 -7186.487,E2 -7186.487} C_VEL
LIN {X 0,Y 474.678,Z 717.359,A -85,B 0,C 180,E1 -7188.903,E2 -7188.903} C_VEL
LIN {X 0,Y 474.716,Z 717.356,A -85,B 0,C 180,E1 -7191.486,E2 -7191.486} C_VEL
LIN {X 0,Y 474.746,Z 717.345,A -85,B 0,C 180,E1 -7194.904,E2 -7194.904} C_VEL
LIN {X 0,Y 474.89,Z 717.333,A -85,B 0,C 180,E1 -7197.455,E2 -7197.455} C_VEL
LIN {X 0,Y 474.915,Z 717.329,A -85,B 0,C 180,E1 -7200,E2 -7200} C_VEL
LIN {X 0,Y 474.891,Z 717.325,A -85,B 0,C 180,E1 -7202.545,E2 -7202.545} C_VEL
LIN {X 0,Y 474.776,Z 717.344,A -85,B 0,C 180,E1 -7205.948,E2 -7205.948} C_VEL
LIN {X 0,Y 474.715,Z 717.346,A -85,B 0,C 180,E1 -7208.514,E2 -7208.514} C_VEL
LIN {X 0,Y 474.709,Z 717.353,A -85,B 0,C 180,E1 -7211.962,E2 -7211.962} C_VEL
LIN {X 0,Y 474.704,Z 717.347,A -85,B 0,C 180,E1 -7215.456,E2 -7215.456} C_VEL
LIN {X 0,Y 474.667,Z 717.355,A -85,B 0,C 180,E1 -7219.01,E2 -7219.01} C_VEL
LIN {X 0,Y 474.592,Z 717.363,A -85,B 0,C 180,E1 -7221.729,E2 -7221.729} C_VEL
LIN {X 0,Y 474.644,Z 717.363,A -85,B 0,C 180,E1 -7224.494,E2 -7224.494} C_VEL
LIN {X 0,Y 474.685,Z 717.353,A -85,B 0,C 180,E1 -7227.334,E2 -7227.334} C_VEL
LIN {X 0,Y 474.61,Z 717.368,A -85,B 0,C 180,E1 -7230.23,E2 -7230.23} C_VEL
LIN {X 0,Y 474.646,Z 717.358,A -85,B 0,C 180,E1 -7233.22,E2 -7233.22} C_VEL
LIN {X 0,Y 474.592,Z 717.372,A -85,B 0,C 180,E1 -7236.323,E2 -7236.323} C_VEL
LIN {X 0,Y 474.631,Z 717.363,A -85,B 0,C 180,E1 -7239.647,E2 -7239.647} C_VEL
LIN {X 0,Y 474.618,Z 717.367,A -85,B 0,C 180,E1 -7242.934,E2 -7242.934} C_VEL
LIN {X 0,Y 474.613,Z 717.365,A -85,B 0,C 180,E1 -7245.895,E2 -7245.895} C_VEL
LIN {X 0,Y 474.631,Z 717.367,A -85,B 0,C 180,E1 -7249.041,E2 -7249.041} C_VEL
LIN {X 0,Y 474.67,Z 717.586,A -85,B 0,C 180,E1 -7249.868,E2 -7249.868} C_VEL
LIN {X 0,Y 476.671,Z 727.737,A -85,B 0,C 180,E1 -7252.807,E2 -7252.807} C_VEL
LIN {X 0,Y 477.063,Z 731.804,A -85,B 0,C 180,E1 -7253.894,E2 -7253.894} C_VEL
LIN {X 0,Y 476.58,Z 744.041,A -85,B 0,C 180,E1 -7256.932,E2 -7256.932} C_VEL
LIN {X 0,Y 476.136,Z 755.419,A -85,B 0,C 180,E1 -7259.632,E2 -7259.632} C_VEL
LIN {X 0,Y 475.768,Z 769.039,A -85,B 0,C 180,E1 -7262.746,E2 -7262.746} C_VEL
LIN {X 0,Y 475.425,Z 782.711,A -85,B 0,C 180,E1 -7265.782,E2 -7265.782} C_VEL
LIN {X 0,Y 475.084,Z 797.45,A -85,B 0,C 180,E1 -7268.971,E2 -7268.971} C_VEL
LIN {X 0,Y 474.779,Z 813.249,A -85,B 0,C 180,E1 -7272.335,E2 -7272.335} C_VEL
LIN {X 0,Y 474.518,Z 824.837,A -85,B 0,C 180,E1 -7274.786,E2 -7274.786} C_VEL
LIN {X 0,Y 475.888,Z 838.557,A -85,B 0,C 180,E1 -7275.159,E2 -7275.159} C_VEL
LIN {X 0,Y 476.856,Z 846.05,A -85,B 0,C 180,E1 -7275.435,E2 -7275.435} C_VEL
LIN {X 0,Y 476.497,Z 858.338,A -85,B 0,C 180,E1 -7275.969,E2 -7275.969} C_VEL
LIN {X 0,Y 475.939,Z 870.747,A -85,B 0,C 180,E1 -7276.693,E2 -7276.693} C_VEL
LIN {X 0,Y 475.51,Z 881.752,A -85,B 0,C 180,E1 -7277.51,E2 -7277.51} C_VEL
LIN {X 0,Y 475.1,Z 892.329,A -85,B 0,C 180,E1 -7278.48,E2 -7278.48} C_VEL
LIN {X 0,Y 474.712,Z 901.778,A -85,B 0,C 180,E1 -7279.551,E2 -7279.551} C_VEL
LIN {X 0,Y 474.409,Z 911.006,A -85,B 0,C 180,E1 -7280.836,E2 -7280.836} C_VEL
LIN {X 0,Y 474.158,Z 918.458,A -85,B 0,C 180,E1 -7282.12,E2 -7282.12} C_VEL
LIN {X 0,Y 474.032,Z 924.361,A -85,B 0,C 180,E1 -7283.387,E2 -7283.387} C_VEL
LIN {X 0,Y 473.976,Z 928.406,A -85,B 0,C 180,E1 -7284.469,E2 -7284.469} C_VEL
LIN {X 0,Y 473.874,Z 932.155,A -85,B 0,C 180,E1 -7285.747,E2 -7285.747} C_VEL
LIN {X 0,Y 473.885,Z 934.106,A -85,B 0,C 180,E1 -7286.599,E2 -7286.599} C_VEL
LIN {X 0,Y 473.845,Z 935.559,A -85,B 0,C 180,E1 -7287.45,E2 -7287.45} C_VEL
LIN {X 0,Y 473.825,Z 936.599,A -85,B 0,C 180,E1 -7288.3,E2 -7288.3} C_VEL
LIN {X 0,Y 473.777,Z 937.238,A -85,B 0,C 180,E1 -7289.15,E2 -7289.15} C_VEL
LIN {X 0,Y 473.763,Z 937.475,A -85,B 0,C 180,E1 -7290,E2 -7290} C_VEL
LIN {X 0,Y 473.774,Z 937.264,A -85,B 0,C 180,E1 -7290.85,E2 -7290.85} C_VEL
LIN {X 0,Y 473.818,Z 936.653,A -85,B 0,C 180,E1 -7291.7,E2 -7291.7} C_VEL
LIN {X 0,Y 473.837,Z 935.641,A -85,B 0,C 180,E1 -7292.55,E2 -7292.55} C_VEL
LIN {X 0,Y 473.885,Z 934.217,A -85,B 0,C 180,E1 -7293.401,E2 -7293.401} C_VEL
LIN {X 0,Y 473.868,Z 931.201,A -85,B 0,C 180,E1 -7294.679,E2 -7294.679} C_VEL
LIN {X 0,Y 474.01,Z 927.137,A -85,B 0,C 180,E1 -7295.957,E2 -7295.957} C_VEL
LIN {X 0,Y 474.098,Z 920.858,A -85,B 0,C 180,E1 -7297.453,E2 -7297.453} C_VEL
LIN {X 0,Y 474.318,Z 914.028,A -85,B 0,C 180,E1 -7298.736,E2 -7298.736} C_VEL
LIN {X 0,Y 474.591,Z 905.572,A -85,B 0,C 180,E1 -7300.02,E2 -7300.02} C_VEL
LIN {X 0,Y 474.979,Z 896.91,A -85,B 0,C 180,E1 -7301.09,E2 -7301.09} C_VEL
LIN {X 0,Y 475.469,Z 886.295,A -85,B 0,C 180,E1 -7302.155,E2 -7302.155} C_VEL
LIN {X 0,Y 475.914,Z 874.719,A -85,B 0,C 180,E1 -7303.091,E2 -7303.091} C_VEL
LIN {X 0,Y 476.277,Z 864.209,A -85,B 0,C 180,E1 -7303.765,E2 -7303.765} C_VEL
LIN {X 0,Y 476.729,Z 852.395,A -85,B 0,C 180,E1 -7304.35,E2 -7304.35} C_VEL
LIN {X 0,Y 476.742,Z 844.018,A -85,B 0,C 180,E1 -7304.677,E2 -7304.677} C_VEL
LIN {X 0,Y 475.118,Z 831.688,A -85,B 0,C 180,E1 -7305.075,E2 -7305.075} C_VEL
LIN {X 0,Y 474.518,Z 825.968,A -85,B 0,C 180,E1 -7305.214,E2 -7305.214} C_VEL
LIN {X 0,Y 474.878,Z 811.354,A -85,B 0,C 180,E1 -7308.407,E2 -7308.407} C_VEL
LIN {X 0,Y 475.247,Z 796.461,A -85,B 0,C 180,E1 -7311.697,E2 -7311.697} C_VEL
LIN {X 0,Y 475.62,Z 784.262,A -85,B 0,C 180,E1 -7314.44,E2 -7314.44} C_VEL
LIN {X 0,Y 476.111,Z 772.107,A -85,B 0,C 180,E1 -7317.232,E2 -7317.232} C_VEL
LIN {X 0,Y 476.658,Z 757.897,A -85,B 0,C 180,E1 -7320.576,E2 -7320.576} C_VEL
LIN {X 0,Y 477.313,Z 744.707,A -85,B 0,C 180,E1 -7323.768,E2 -7323.768} C_VEL
LIN {X 0,Y 477.814,Z 733.575,A -85,B 0,C 180,E1 -7326.563,E2 -7326.563} C_VEL
LIN {X 0,Y 476.452,Z 726.254,A -85,B 0,C 180,E1 -7328.575,E2 -7328.575} C_VEL
LIN {X 0,Y 474.653,Z 717.363,A -85,B 0,C 180,E1 -7331.172,E2 -7331.172} C_VEL
LIN {X 0,Y 474.612,Z 717.364,A -85,B 0,C 180,E1 -7334.105,E2 -7334.105} C_VEL
LIN {X 0,Y 474.617,Z 717.366,A -85,B 0,C 180,E1 -7337.066,E2 -7337.066} C_VEL
LIN {X 0,Y 474.647,Z 717.356,A -85,B 0,C 180,E1 -7340.454,E2 -7340.454} C_VEL
LIN {X 0,Y 474.591,Z 717.37,A -85,B 0,C 180,E1 -7343.677,E2 -7343.677} C_VEL
LIN {X 0,Y 474.645,Z 717.357,A -85,B 0,C 180,E1 -7346.78,E2 -7346.78} C_VEL
LIN {X 0,Y 474.608,Z 717.368,A -85,B 0,C 180,E1 -7349.77,E2 -7349.77} C_VEL
LIN {X 0,Y 474.699,Z 717.35,A -85,B 0,C 180,E1 -7352.68,E2 -7352.68} C_VEL
LIN {X 0,Y 474.643,Z 717.362,A -85,B 0,C 180,E1 -7355.506,E2 -7355.506} C_VEL
LIN {X 0,Y 474.673,Z 717.356,A -85,B 0,C 180,E1 -7359.185,E2 -7359.185} C_VEL
LIN {X 0,Y 474.649,Z 717.364,A -85,B 0,C 180,E1 -7361.884,E2 -7361.884} C_VEL
LIN {X 0,Y 474.703,Z 717.351,A -85,B 0,C 180,E1 -7364.544,E2 -7364.544} C_VEL
LIN {X 0,Y 474.708,Z 717.357,A -85,B 0,C 180,E1 -7368.038,E2 -7368.038} C_VEL
LIN {X 0,Y 474.729,Z 717.35,A -85,B 0,C 180,E1 -7371.487,E2 -7371.487} C_VEL
LIN {X 0,Y 474.774,Z 717.347,A -85,B 0,C 180,E1 -7374.052,E2 -7374.052} C_VEL
LIN {X 0,Y 474.886,Z 717.329,A -85,B 0,C 180,E1 -7377.455,E2 -7377.455} C_VEL
LIN {X 0,Y 474.913,Z 717.328,A -85,B 0,C 180,E1 -7380,E2 -7380} C_VEL
LIN {X 0,Y 474.888,Z 717.332,A -85,B 0,C 180,E1 -7382.545,E2 -7382.545} C_VEL
LIN {X 0,Y 474.757,Z 717.347,A -85,B 0,C 180,E1 -7385.948,E2 -7385.948} C_VEL
LIN {X 0,Y 474.714,Z 717.355,A -85,B 0,C 180,E1 -7388.514,E2 -7388.514} C_VEL
LIN {X 0,Y 474.707,Z 717.354,A -85,B 0,C 180,E1 -7391.962,E2 -7391.962} C_VEL
LIN {X 0,Y 474.701,Z 717.352,A -85,B 0,C 180,E1 -7395.456,E2 -7395.456} C_VEL
LIN {X 0,Y 474.664,Z 717.358,A -85,B 0,C 180,E1 -7399.01,E2 -7399.01} C_VEL
LIN {X 0,Y 474.591,Z 717.366,A -85,B 0,C 180,E1 -7401.729,E2 -7401.729} C_VEL
LIN {X 0,Y 474.627,Z 717.364,A -85,B 0,C 180,E1 -7404.495,E2 -7404.495} C_VEL
LIN {X 0,Y 474.639,Z 717.36,A -85,B 0,C 180,E1 -7407.324,E2 -7407.324} C_VEL
LIN {X 0,Y 474.604,Z 717.367,A -85,B 0,C 180,E1 -7410.231,E2 -7410.231} C_VEL
LIN {X 0,Y 474.617,Z 717.364,A -85,B 0,C 180,E1 -7413.222,E2 -7413.222} C_VEL
LIN {X 0,Y 474.582,Z 717.37,A -85,B 0,C 180,E1 -7416.324,E2 -7416.324} C_VEL
LIN {X 0,Y 474.602,Z 717.364,A -85,B 0,C 180,E1 -7419.644,E2 -7419.644} C_VEL
LIN {X 0,Y 474.571,Z 717.371,A -85,B 0,C 180,E1 -7422.94,E2 -7422.94} C_VEL
LIN {X 0,Y 474.603,Z 717.364,A -85,B 0,C 180,E1 -7425.894,E2 -7425.894} C_VEL
LIN {X 0,Y 474.592,Z 717.369,A -85,B 0,C 180,E1 -7429.34,E2 -7429.34} C_VEL
LIN {X 0,Y 474.592,Z 717.366,A -85,B 0,C 180,E1 -7431.707,E2 -7431.707} C_VEL
LIN {X 0,Y 474.612,Z 717.367,A -85,B 0,C 180,E1 -7434.725,E2 -7434.725} C_VEL
LIN {X 0,Y 474.612,Z 717.364,A -85,B 0,C 180,E1 -7437.786,E2 -7437.786} C_VEL
LIN {X 0,Y 474.595,Z 717.37,A -85,B 0,C 180,E1 -7440.892,E2 -7440.892} C_VEL
LIN {X 0,Y 474.573,Z 717.371,A -85,B 0,C 180,E1 -7443.623,E2 -7443.623} C_VEL
LIN {X 0,Y 474.636,Z 717.361,A -85,B 0,C 180,E1 -7446.642,E2 -7446.642} C_VEL
LIN {X 0,Y 474.654,Z 717.358,A -85,B 0,C 180,E1 -7450.09,E2 -7450.09} C_VEL
LIN {X 0,Y 474.646,Z 717.361,A -85,B 0,C 180,E1 -7451.655,E2 -7451.655} C_VEL
LIN {X 0,Y 473.973,Z 717.445,A -85,B 0,C 180,E1 -7452.364,E2 -7452.364} C_VEL
LIN {X 0,Y 471.125,Z 717.804,A -85,B 0,C 180,E1 -7453.515,E2 -7453.515} C_VEL
LIN {X 0,Y 468.717,Z 718.105,A -85,B 0,C 180,E1 -7454.443,E2 -7454.443} C_VEL
LIN {X 0,Y 467.678,Z 718.231,A -85,B 0,C 180,E1 -7455.16,E2 -7455.16} C_VEL
LIN {X 0,Y 467.591,Z 718.24,A -85,B 0,C 180,E1 -7455.403,E2 -7455.403} C_VEL
LIN {X 0,Y 467.65,Z 718.232,A -85,B 0,C 180,E1 -7457.854,E2 -7457.854} C_VEL
LIN {X 0,Y 467.632,Z 718.237,A -85,B 0,C 180,E1 -7461.356,E2 -7461.356} C_VEL
LIN {X 0,Y 467.703,Z 718.225,A -85,B 0,C 180,E1 -7463.962,E2 -7463.962} C_VEL
LIN {X 0,Y 467.814,Z 718.215,A -85,B 0,C 180,E1 -7467.417,E2 -7467.417} C_VEL
LIN {X 0,Y 467.852,Z 718.207,A -85,B 0,C 180,E1 -7470,E2 -7470} C_VEL
LIN {X 0,Y 467.816,Z 718.209,A -85,B 0,C 180,E1 -7472.583,E2 -7472.583} C_VEL
LIN {X 0,Y 467.707,Z 718.225,A -85,B 0,C 180,E1 -7476.038,E2 -7476.038} C_VEL
LIN {X 0,Y 467.661,Z 718.228,A -85,B 0,C 180,E1 -7478.643,E2 -7478.643} C_VEL
LIN {X 0,Y 467.66,Z 718.231,A -85,B 0,C 180,E1 -7482.145,E2 -7482.145} C_VEL
LIN {X 0,Y 467.643,Z 718.235,A -85,B 0,C 180,E1 -7485.695,E2 -7485.695} C_VEL
LIN {X 0,Y 467.625,Z 718.233,A -85,B 0,C 180,E1 -7489.308,E2 -7489.308} C_VEL
LIN {X 0,Y 467.539,Z 718.249,A -85,B 0,C 180,E1 -7492.074,E2 -7492.074} C_VEL
LIN {X 0,Y 467.571,Z 718.239,A -85,B 0,C 180,E1 -7494.889,E2 -7494.889} C_VEL
LIN {X 0,Y 467.582,Z 718.24,A -85,B 0,C 180,E1 -7497.772,E2 -7497.772} C_VEL
LIN {X 0,Y 467.571,Z 718.239,A -85,B 0,C 180,E1 -7501.045,E2 -7501.045} C_VEL
LIN {X 0,Y 467.581,Z 718.245,A -85,B 0,C 180,E1 -7504.24,E2 -7504.24} C_VEL
LIN {X 0,Y 467.552,Z 718.241,A -85,B 0,C 180,E1 -7507.186,E2 -7507.186} C_VEL
LIN {X 0,Y 467.578,Z 718.244,A -85,B 0,C 180,E1 -7510.265,E2 -7510.265} C_VEL
LIN {X 0,Y 467.59,Z 718.242,A -85,B 0,C 180,E1 -7512.567,E2 -7512.567} C_VEL
LIN {X 0,Y 467.57,Z 718.241,A -85,B 0,C 180,E1 -7515.053,E2 -7515.053} C_VEL
LIN {X 0,Y 467.592,Z 718.239,A -85,B 0,C 180,E1 -7517.522,E2 -7517.522} C_VEL
LIN {X 0,Y 470.226,Z 727.794,A -85,B 0,C 180,E1 -7518.116,E2 -7518.116} C_VEL
LIN {X 0,Y 469.928,Z 739.037,A -85,B 0,C 180,E1 -7518.849,E2 -7518.849} C_VEL
LIN {X 0,Y 469.471,Z 750.191,A -85,B 0,C 180,E1 -7519.772,E2 -7519.772} C_VEL
LIN {X 0,Y 469.104,Z 760.789,A -85,B 0,C 180,E1 -7520.868,E2 -7520.868} C_VEL
LIN {X 0,Y 468.664,Z 770.046,A -85,B 0,C 180,E1 -7522.06,E2 -7522.06} C_VEL
LIN {X 0,Y 468.248,Z 778.262,A -85,B 0,C 180,E1 -7523.372,E2 -7523.372} C_VEL
LIN {X 0,Y 467.977,Z 784.846,A -85,B 0,C 180,E1 -7524.682,E2 -7524.682} C_VEL
LIN {X 0,Y 467.665,Z 790.84,A -85,B 0,C 180,E1 -7526.218,E2 -7526.218} C_VEL
LIN {X 0,Y 467.538,Z 795.366,A -85,B 0,C 180,E1 -7527.793,E2 -7527.793} C_VEL
LIN {X 0,Y 467.379,Z 798.267,A -85,B 0,C 180,E1 -7529.252,E2 -7529.252} C_VEL
LIN {X 0,Y 467.321,Z 799.973,A -85,B 0,C 180,E1 -7530.723,E2 -7530.723} C_VEL
LIN {X 0,Y 467.291,Z 800.496,A -85,B 0,C 180,E1 -7532.543,E2 -7532.543} C_VEL
LIN {X 0,Y 467.365,Z 799.529,A -85,B 0,C 180,E1 -7534.145,E2 -7534.145} C_VEL
LIN {X 0,Y 467.474,Z 798.255,A -85,B 0,C 180,E1 -7535.105,E2 -7535.105} C_VEL
LIN {X 0,Y 467.651,Z 795.635,A -85,B 0,C 180,E1 -7536.453,E2 -7536.453} C_VEL
LIN {X 0,Y 467.839,Z 791.506,A -85,B 0,C 180,E1 -7537.941,E2 -7537.941} C_VEL
LIN {X 0,Y 468.12,Z 786.277,A -85,B 0,C 180,E1 -7539.34,E2 -7539.34} C_VEL
LIN {X 0,Y 468.487,Z 779.551,A -85,B 0,C 180,E1 -7540.729,E2 -7540.729} C_VEL
LIN {X 0,Y 468.893,Z 771.161,A -85,B 0,C 180,E1 -7542.105,E2 -7542.105} C_VEL
LIN {X 0,Y 469.345,Z 762.229,A -85,B 0,C 180,E1 -7543.269,E2 -7543.269} C_VEL
LIN {X 0,Y 469.783,Z 751.653,A -85,B 0,C 180,E1 -7544.378,E2 -7544.378} C_VEL
LIN {X 0,Y 470.206,Z 740.865,A -85,B 0,C 180,E1 -7545.28,E2 -7545.28} C_VEL
LIN {X 0,Y 470.501,Z 728.874,A -85,B 0,C 180,E1 -7546.062,E2 -7546.062} C_VEL
LIN {X 0,Y 467.624,Z 718.236,A -85,B 0,C 180,E1 -7546.75,E2 -7546.75} C_VEL
LIN {X 0,Y 467.626,Z 718.241,A -85,B 0,C 180,E1 -7549.61,E2 -7549.61} C_VEL
LIN {X 0,Y 467.697,Z 718.223,A -85,B 0,C 180,E1 -7552.647,E2 -7552.647} C_VEL
LIN {X 0,Y 467.717,Z 718.22,A -85,B 0,C 180,E1 -7554.827,E2 -7554.827} C_VEL
LIN {X 0,Y 467.855,Z 718.208,A -85,B 0,C 180,E1 -7557.417,E2 -7557.417} C_VEL
LIN {X 0,Y 467.885,Z 718.205,A -85,B 0,C 180,E1 -7560,E2 -7560} C_VEL
LIN {X 0,Y 467.856,Z 718.201,A -85,B 0,C 180,E1 -7562.583,E2 -7562.583} C_VEL
LIN {X 0,Y 467.74,Z 718.22,A -85,B 0,C 180,E1 -7566.037,E2 -7566.037} C_VEL
LIN {X 0,Y 467.673,Z 718.223,A -85,B 0,C 180,E1 -7568.643,E2 -7568.643} C_VEL
LIN {X 0,Y 467.66,Z 718.23,A -85,B 0,C 180,E1 -7572.145,E2 -7572.145} C_VEL
LIN {X 0,Y 467.643,Z 718.229,A -85,B 0,C 180,E1 -7575.695,E2 -7575.695} C_VEL
LIN {X 0,Y 467.617,Z 718.234,A -85,B 0,C 180,E1 -7578.763,E2 -7578.763} C_VEL
LIN {X 0,Y 467.584,Z 718.234,A -85,B 0,C 180,E1 -7581.268,E2 -7581.268} C_VEL
LIN {X 0,Y 467.567,Z 718.242,A -85,B 0,C 180,E1 -7583.944,E2 -7583.944} C_VEL
LIN {X 0,Y 467.617,Z 718.236,A -85,B 0,C 180,E1 -7586.8,E2 -7586.8} C_VEL
LIN {X 0,Y 467.558,Z 718.241,A -85,B 0,C 180,E1 -7589.738,E2 -7589.738} C_VEL
LIN {X 0,Y 467.587,Z 718.24,A -85,B 0,C 180,E1 -7592.758,E2 -7592.758} C_VEL
LIN {X 0,Y 467.557,Z 718.243,A -85,B 0,C 180,E1 -7595.889,E2 -7595.889} C_VEL
LIN {X 0,Y 467.586,Z 718.243,A -85,B 0,C 180,E1 -7599.144,E2 -7599.144} C_VEL
LIN {X 0,Y 467.589,Z 718.245,A -85,B 0,C 180,E1 -7602.567,E2 -7602.567} C_VEL
LIN {X 0,Y 467.574,Z 718.243,A -85,B 0,C 180,E1 -7605.053,E2 -7605.053} C_VEL
LIN {X 0,Y 467.592,Z 718.243,A -85,B 0,C 180,E1 -7607.44,E2 -7607.44} C_VEL
LIN {X 0,Y 467.636,Z 718.393,A -85,B 0,C 180,E1 -7609.529,E2 -7609.529} C_VEL
LIN {X 0,Y 469.569,Z 728.321,A -85,B 0,C 180,E1 -7612.49,E2 -7612.49} C_VEL
LIN {X 0,Y 470.118,Z 733.174,A -85,B 0,C 180,E1 -7613.83,E2 -7613.83} C_VEL
LIN {X 0,Y 469.568,Z 745.485,A -85,B 0,C 180,E1 -7616.945,E2 -7616.945} C_VEL
LIN {X 0,Y 469.123,Z 756.578,A -85,B 0,C 180,E1 -7619.628,E2 -7619.628} C_VEL
LIN {X 0,Y 468.726,Z 770.13,A -85,B 0,C 180,E1 -7622.786,E2 -7622.786} C_VEL
LIN {X 0,Y 468.361,Z 783.776,A -85,B 0,C 180,E1 -7625.864,E2 -7625.864} C_VEL
LIN {X 0,Y 467.937,Z 799.524,A -85,B 0,C 180,E1 -7629.332,E2 -7629.332} C_VEL
LIN {X 0,Y 467.659,Z 814.157,A -85,B 0,C 180,E1 -7632.509,E2 -7632.509} C_VEL
LIN {X 0,Y 467.462,Z 823.653,A -85,B 0,C 180,E1 -7634.55,E2 -7634.55} C_VEL
LIN {X 0,Y 468.854,Z 838.626,A -85,B 0,C 180,E1 -7634.973,E2 -7634.973} C_VEL
LIN {X 0,Y 469.916,Z 847.587,A -85,B 0,C 180,E1 -7635.326,E2 -7635.326} C_VEL
LIN {X 0,Y 469.413,Z 860.107,A -85,B 0,C 180,E1 -7635.919,E2 -7635.919} C_VEL
LIN {X 0,Y 468.868,Z 872.249,A -85,B 0,C 180,E1 -7636.676,E2 -7636.676} C_VEL
LIN {X 0,Y 468.452,Z 882.94,A -85,B 0,C 180,E1 -7637.524,E2 -7637.524} C_VEL
LIN {X 0,Y 468.031,Z 894.184,A -85,B 0,C 180,E1 -7638.633,E2 -7638.633} C_VEL
LIN {X 0,Y 467.558,Z 903.962,A -85,B 0,C 180,E1 -7639.827,E2 -7639.827} C_VEL
LIN {X 0,Y 467.257,Z 912.532,A -85,B 0,C 180,E1 -7641.131,E2 -7641.131} C_VEL
LIN {X 0,Y 467.061,Z 919.471,A -85,B 0,C 180,E1 -7642.434,E2 -7642.434} C_VEL
LIN {X 0,Y 466.969,Z 925.854,A -85,B 0,C 180,E1 -7643.952,E2 -7643.952} C_VEL
LIN {X 0,Y 466.844,Z 929.991,A -85,B 0,C 180,E1 -7645.25,E2 -7645.25} C_VEL
LIN {X 0,Y 466.845,Z 933.067,A -85,B 0,C 180,E1 -7646.548,E2 -7646.548} C_VEL
LIN {X 0,Y 466.809,Z 934.529,A -85,B 0,C 180,E1 -7647.411,E2 -7647.411} C_VEL
LIN {X 0,Y 466.792,Z 935.575,A -85,B 0,C 180,E1 -7648.274,E2 -7648.274} C_VEL
LIN {X 0,Y 466.749,Z 936.225,A -85,B 0,C 180,E1 -7649.137,E2 -7649.137} C_VEL
LIN {X 0,Y 466.736,Z 936.468,A -85,B 0,C 180,E1 -7650,E2 -7650} C_VEL
LIN {X 0,Y 466.744,Z 936.26,A -85,B 0,C 180,E1 -7650.863,E2 -7650.863} C_VEL
LIN {X 0,Y 466.783,Z 935.652,A -85,B 0,C 180,E1 -7651.725,E2 -7651.725} C_VEL
LIN {X 0,Y 466.797,Z 934.646,A -85,B 0,C 180,E1 -7652.589,E2 -7652.589} C_VEL
LIN {X 0,Y 466.845,Z 933.223,A -85,B 0,C 180,E1 -7653.452,E2 -7653.452} C_VEL
LIN {X 0,Y 466.83,Z 930.211,A -85,B 0,C 180,E1 -7654.75,E2 -7654.75} C_VEL
LIN {X 0,Y 466.93,Z 925.2,A -85,B 0,C 180,E1 -7656.298,E2 -7656.298} C_VEL
LIN {X 0,Y 467.048,Z 918.829,A -85,B 0,C 180,E1 -7657.783,E2 -7657.783} C_VEL
LIN {X 0,Y 467.282,Z 911.77,A -85,B 0,C 180,E1 -7659.086,E2 -7659.086} C_VEL
LIN {X 0,Y 467.592,Z 902.932,A -85,B 0,C 180,E1 -7660.391,E2 -7660.391} C_VEL
LIN {X 0,Y 468.036,Z 893.921,A -85,B 0,C 180,E1 -7661.476,E2 -7661.476} C_VEL
LIN {X 0,Y 468.531,Z 883.509,A -85,B 0,C 180,E1 -7662.503,E2 -7662.503} C_VEL
LIN {X 0,Y 468.904,Z 873.257,A -85,B 0,C 180,E1 -7663.323,E2 -7663.323} C_VEL
LIN {X 0,Y 469.434,Z 861.219,A -85,B 0,C 180,E1 -7664.08,E2 -7664.08} C_VEL
LIN {X 0,Y 469.907,Z 848.805,A -85,B 0,C 180,E1 -7664.674,E2 -7664.674} C_VEL
LIN {X 0,Y 469.682,Z 844.122,A -85,B 0,C 180,E1 -7664.861,E2 -7664.861} C_VEL
LIN {X 0,Y 468.228,Z 832.492,A -85,B 0,C 180,E1 -7665.256,E2 -7665.256} C_VEL
LIN {X 0,Y 467.463,Z 825.058,A -85,B 0,C 180,E1 -7665.45,E2 -7665.45} C_VEL
LIN {X 0,Y 467.789,Z 811.851,A -85,B 0,C 180,E1 -7668.391,E2 -7668.391} C_VEL
LIN {X 0,Y 468.185,Z 797.157,A -85,B 0,C 180,E1 -7671.7,E2 -7671.7} C_VEL
LIN {X 0,Y 468.655,Z 783.519,A -85,B 0,C 180,E1 -7674.828,E2 -7674.828} C_VEL
LIN {X 0,Y 469.18,Z 770.427,A -85,B 0,C 180,E1 -7677.898,E2 -7677.898} C_VEL
LIN {X 0,Y 469.751,Z 757.318,A -85,B 0,C 180,E1 -7681.045,E2 -7681.045} C_VEL
LIN {X 0,Y 470.417,Z 745.087,A -85,B 0,C 180,E1 -7684.073,E2 -7684.073} C_VEL
LIN {X 0,Y 470.883,Z 734.931,A -85,B 0,C 180,E1 -7686.656,E2 -7686.656} C_VEL
LIN {X 0,Y 469.292,Z 726.662,A -85,B 0,C 180,E1 -7688.975,E2 -7688.975} C_VEL
LIN {X 0,Y 467.603,Z 718.241,A -85,B 0,C 180,E1 -7691.472,E2 -7691.472} C_VEL
LIN {X 0,Y 467.573,Z 718.244,A -85,B 0,C 180,E1 -7695.053,E2 -7695.053} C_VEL
LIN {X 0,Y 467.591,Z 718.243,A -85,B 0,C 180,E1 -7697.44,E2 -7697.44} C_VEL
LIN {X 0,Y 467.585,Z 718.238,A -85,B 0,C 180,E1 -7700.855,E2 -7700.855} C_VEL
LIN {X 0,Y 467.562,Z 718.24,A -85,B 0,C 180,E1 -7704.261,E2 -7704.261} C_VEL
LIN {X 0,Y 467.584,Z 718.24,A -85,B 0,C 180,E1 -7707.321,E2 -7707.321} C_VEL
LIN {X 0,Y 467.572,Z 718.238,A -85,B 0,C 180,E1 -7710.667,E2 -7710.667} C_VEL
LIN {X 0,Y 467.615,Z 718.235,A -85,B 0,C 180,E1 -7713.2,E2 -7713.2} C_VEL
LIN {X 0,Y 467.593,Z 718.236,A -85,B 0,C 180,E1 -7716.469,E2 -7716.469} C_VEL
LIN {X 0,Y 467.625,Z 718.238,A -85,B 0,C 180,E1 -7719.777,E2 -7719.777} C_VEL
LIN {X 0,Y 467.601,Z 718.236,A -85,B 0,C 180,E1 -7722.506,E2 -7722.506} C_VEL
LIN {X 0,Y 467.609,Z 718.235,A -85,B 0,C 180,E1 -7725.197,E2 -7725.197} C_VEL
LIN {X 0,Y 467.659,Z 718.232,A -85,B 0,C 180,E1 -7727.855,E2 -7727.855} C_VEL
LIN {X 0,Y 467.683,Z 718.227,A -85,B 0,C 180,E1 -7731.357,E2 -7731.357} C_VEL
LIN {X 0,Y 467.739,Z 718.222,A -85,B 0,C 180,E1 -7733.963,E2 -7733.963} C_VEL
LIN {X 0,Y 467.851,Z 718.206,A -85,B 0,C 180,E1 -7737.417,E2 -7737.417} C_VEL
LIN {X 0,Y 467.883,Z 718.204,A -85,B 0,C 180,E1 -7740,E2 -7740} C_VEL
LIN {X 0,Y 467.853,Z 718.208,A -85,B 0,C 180,E1 -7742.583,E2 -7742.583} C_VEL
LIN {X 0,Y 467.72,Z 718.224,A -85,B 0,C 180,E1 -7746.038,E2 -7746.038} C_VEL
LIN {X 0,Y 467.672,Z 718.231,A -85,B 0,C 180,E1 -7748.643,E2 -7748.643} C_VEL
LIN {X 0,Y 467.659,Z 718.232,A -85,B 0,C 180,E1 -7752.146,E2 -7752.146} C_VEL
